(* IEC 61131-3 sources: TIA2AX/tests/V18/test_projects/expected/HW_2000528_ST43/PLC_4.3, 7 files *)

(* ---- HwIdentifiers.st ---- *)
TYPE
	HwIdentifiers : WORD
	(
		PLC_4_3_Rail_0 :=	WORD#256,
		PLC_4_3 :=	WORD#48,
		PLC_4_3_Card_reader_writer_1 :=	WORD#51,
		PLC_4_3_CPU_display_1 :=	WORD#54,
		PLC_4_3_OPC_UA_1 :=	WORD#117,
		PLC_4_3_PROFINET_interface_1 :=	WORD#64,
		PLC_4_3_PROFINET_interface_1_Port_1 :=	WORD#65,
		PLC_4_3_PROFINET_interface_1_Port_2 :=	WORD#66,
		PLC_4_3_PROFINET_interface_2 :=	WORD#72,
		PLC_4_3_PROFINET_interface_2_Port_1 :=	WORD#73,
		wp4_3_dm262_l_Rack :=	WORD#270,
		wp4_3_dm262_l :=	WORD#258,
		wp4_3_dm262_l_Interface :=	WORD#259,
		wp4_3_dm262_l_Interface_Port_1 :=	WORD#260,
		wp4_3_dm262_l_DataMan_260 :=	WORD#261,
		wp4_3_dm262_l_Acquisition_Control_1 :=	WORD#262,
		wp4_3_dm262_l_Acquisition_Status_1 :=	WORD#263,
		wp4_3_dm262_l_Results_Control_1 :=	WORD#264,
		wp4_3_dm262_l_Results_Status_1 :=	WORD#265,
		wp4_3_dm262_l_Soft_Event_Control_1 :=	WORD#266,
		wp4_3_dm262_l_User_Data_64_bytes_1 :=	WORD#267,
		wp4_3_dm262_l_Result_Data_64_bytes_1 :=	WORD#268,
		ET_200SP_ST43_Rack_0 :=	WORD#278,
		ET_200SP_ST43 :=	WORD#279,
		ET_200SP_ST43_ET_200SP_ST43 :=	WORD#280,
		ET_200SP_ST43_PROFINET_interface :=	WORD#281,
		ET_200SP_ST43_PROFINET_interface_Port_1 :=	WORD#283,
		ET_200SP_ST43_PROFINET_interface_Port_2 :=	WORD#282,
		ET_200SP_ST43_BA_2xRJ45 :=	WORD#283,
		ET_200SP_ST43_A3 :=	WORD#284,
		ET_200SP_ST43_A4 :=	WORD#285,
		ET_200SP_ST43_A5 :=	WORD#286,
		ET_200SP_ST43_DI_16x24VDC_ST_1 :=	WORD#287,
		ET_200SP_ST43_DI_16x24VDC_ST_2 :=	WORD#288,
		ET_200SP_ST43_DI_16x24VDC_ST_3 :=	WORD#289,
		ET_200SP_ST43_DI_16x24VDC_ST_4 :=	WORD#290,
		ET_200SP_ST43_DQ_16x24VDC_0_5A_ST_1 :=	WORD#291,
		ET_200SP_ST43_DQ_16x24VDC_0_5A_ST_2 :=	WORD#292,
		ET_200SP_ST43_TM_Pulse_2x24V_1 :=	WORD#271,
		ET_200SP_ST43_TM_Pulse_2x24V_2 :=	WORD#272,
		ET_200SP_ST43_TM_Pulse_2x24V_3 :=	WORD#273,
		ET_200SP_ST43_TM_Pulse_2x24V_4 :=	WORD#274,
		ET_200SP_ST43_TM_Pulse_2x24V_5 :=	WORD#275,
		ET_200SP_ST43_Server_module_1 :=	WORD#276,
		wp4_3_dm262_r_Rack :=	WORD#294,
		wp4_3_dm262_r :=	WORD#295,
		wp4_3_dm262_r_Interface :=	WORD#296,
		wp4_3_dm262_r_Interface_Port_1 :=	WORD#297,
		wp4_3_dm262_r_DataMan_260 :=	WORD#298,
		wp4_3_dm262_r_Acquisition_Control_1 :=	WORD#299,
		wp4_3_dm262_r_Acquisition_Status_1 :=	WORD#300,
		wp4_3_dm262_r_Results_Control_1 :=	WORD#301,
		wp4_3_dm262_r_Results_Status_1 :=	WORD#302,
		wp4_3_dm262_r_Soft_Event_Control_1 :=	WORD#303,
		wp4_3_dm262_r_User_Data_64_bytes_1 :=	WORD#304,
		wp4_3_dm262_r_Result_Data_64_bytes_1 :=	WORD#305,
		CPX_ST43_PN_IO_Interface :=	WORD#309,
		CPX_ST43_PN_IO_Interface_Port_1 :=	WORD#310,
		CPX_ST43_PN_IO_Interface_Port_2 :=	WORD#311,
		CPX_ST43_CPX_Rev_30 :=	WORD#312,
		CPX_ST43_FB33_PNIO_Module_1 :=	WORD#313,
		CPX_ST43_MPA1S_VMPA1_FB_EMS_8_8DO_1 :=	WORD#314,
		CPX_ST43_MPA1G_VMPA1_FB_EMG_8_8DO_1 :=	WORD#315,
		CPX_ST43_MPA1G_VMPA1_FB_EMG_8_8DO_2 :=	WORD#316,
		CPX_ST43_MPA1G_VMPA1_FB_EMG_8_8DO_3 :=	WORD#317,
		CPX_ST43_MPA1G_VMPA1_FB_EMG_8_8DO_4 :=	WORD#318,
		CPX_ST43_MPA1G_VMPA1_FB_EMG_8_8DO_5 :=	WORD#319,
		NONE:= WORD#0
	);
END_TYPE

(* ---- HwInputs.st ---- *)
TYPE
	HwInputs : STRUCT
		wp4_3_dm262_l_Acquisition_Status_1 AT %B317 : ARRAY[0..2] OF BYTE;
		wp4_3_dm262_l_Results_Status_1 AT %B301 : BYTE;
		wp4_3_dm262_l_Soft_Event_Control_1 AT %B302 : BYTE;
		wp4_3_dm262_l_Result_Data_64_bytes_1 AT %B503 : ARRAY[0..71] OF BYTE;
		ET_200SP_ST43_A3 AT %B88 : ARRAY[0..7] OF BYTE;
		ET_200SP_ST43_A4 AT %B96 : ARRAY[0..7] OF BYTE;
		ET_200SP_ST43_A5 AT %B104 : ARRAY[0..7] OF BYTE;
		ET_200SP_ST43_DI_16x24VDC_ST_1 AT %B0 : WORD;
		ET_200SP_ST43_DI_16x24VDC_ST_2 AT %B2 : WORD;
		ET_200SP_ST43_DI_16x24VDC_ST_3 AT %B4 : WORD;
		ET_200SP_ST43_DI_16x24VDC_ST_4 AT %B6 : WORD;
		ET_200SP_ST43_TM_Pulse_2x24V_1 AT %B8 : ARRAY[0..15] OF BYTE;
		ET_200SP_ST43_TM_Pulse_2x24V_2 AT %B24 : ARRAY[0..15] OF BYTE;
		ET_200SP_ST43_TM_Pulse_2x24V_3 AT %B40 : ARRAY[0..15] OF BYTE;
		ET_200SP_ST43_TM_Pulse_2x24V_4 AT %B56 : ARRAY[0..15] OF BYTE;
		ET_200SP_ST43_TM_Pulse_2x24V_5 AT %B72 : ARRAY[0..15] OF BYTE;
		wp4_3_dm262_r_Acquisition_Status_1 AT %B281 : ARRAY[0..2] OF BYTE;
		wp4_3_dm262_r_Results_Status_1 AT %B207 : BYTE;
		wp4_3_dm262_r_Soft_Event_Control_1 AT %B208 : BYTE;
		wp4_3_dm262_r_Result_Data_64_bytes_1 AT %B209 : ARRAY[0..71] OF BYTE;
	END_STRUCT;
END_TYPE

(* ---- HwOutputs.st ---- *)
TYPE
	HwOutputs : STRUCT
		wp4_3_dm262_l_Acquisition_Control_1 AT %B300 : BYTE;
		wp4_3_dm262_l_Results_Control_1 AT %B301 : BYTE;
		wp4_3_dm262_l_Soft_Event_Control_1 AT %B302 : BYTE;
		wp4_3_dm262_l_User_Data_64_bytes_1 AT %B303 : ARRAY[0..67] OF BYTE;
		ET_200SP_ST43_DQ_16x24VDC_0_5A_ST_1 AT %B0 : WORD;
		ET_200SP_ST43_DQ_16x24VDC_0_5A_ST_2 AT %B2 : WORD;
		ET_200SP_ST43_TM_Pulse_2x24V_1 AT %B4 : ARRAY[0..23] OF BYTE;
		ET_200SP_ST43_TM_Pulse_2x24V_2 AT %B56 : ARRAY[0..23] OF BYTE;
		ET_200SP_ST43_TM_Pulse_2x24V_3 AT %B80 : ARRAY[0..23] OF BYTE;
		ET_200SP_ST43_TM_Pulse_2x24V_4 AT %B104 : ARRAY[0..23] OF BYTE;
		ET_200SP_ST43_TM_Pulse_2x24V_5 AT %B128 : ARRAY[0..23] OF BYTE;
		wp4_3_dm262_r_Acquisition_Control_1 AT %B400 : BYTE;
		wp4_3_dm262_r_Results_Control_1 AT %B401 : BYTE;
		wp4_3_dm262_r_Soft_Event_Control_1 AT %B402 : BYTE;
		wp4_3_dm262_r_User_Data_64_bytes_1 AT %B403 : ARRAY[0..67] OF BYTE;
		CPX_ST43_MPA1S_VMPA1_FB_EMS_8_8DO_1 AT %B50 : BYTE;
		CPX_ST43_MPA1G_VMPA1_FB_EMG_8_8DO_1 AT %B51 : BYTE;
		CPX_ST43_MPA1G_VMPA1_FB_EMG_8_8DO_2 AT %B52 : BYTE;
		CPX_ST43_MPA1G_VMPA1_FB_EMG_8_8DO_3 AT %B53 : BYTE;
		CPX_ST43_MPA1G_VMPA1_FB_EMG_8_8DO_4 AT %B54 : BYTE;
		CPX_ST43_MPA1G_VMPA1_FB_EMG_8_8DO_5 AT %B55 : BYTE;
	END_STRUCT;
END_TYPE

(* ---- PlcInputs.st ---- *)
TYPE
	PlcInputs : STRUCT
		wp4_3_dm262_l_Acquisition_Status_1 : ARRAY[0..2] OF BYTE;
		wp4_3_dm262_l_Results_Status_1 : BYTE;
		wp4_3_dm262_l_Soft_Event_Control_1 : BYTE;
		wp4_3_dm262_l_Result_Data_64_bytes_1 : ARRAY[0..71] OF BYTE;
		ET_200SP_ST43_A3 : ARRAY[0..7] OF BYTE;
		ET_200SP_ST43_A4 : ARRAY[0..7] OF BYTE;
		ET_200SP_ST43_A5 : ARRAY[0..7] OF BYTE;
		ET_200SP_ST43_DI_16x24VDC_ST_1 : WORD;
		ET_200SP_ST43_DI_16x24VDC_ST_2 : WORD;
		ET_200SP_ST43_DI_16x24VDC_ST_3 : WORD;
		ET_200SP_ST43_DI_16x24VDC_ST_4 : WORD;
		ET_200SP_ST43_TM_Pulse_2x24V_1 : ARRAY[0..15] OF BYTE;
		ET_200SP_ST43_TM_Pulse_2x24V_2 : ARRAY[0..15] OF BYTE;
		ET_200SP_ST43_TM_Pulse_2x24V_3 : ARRAY[0..15] OF BYTE;
		ET_200SP_ST43_TM_Pulse_2x24V_4 : ARRAY[0..15] OF BYTE;
		ET_200SP_ST43_TM_Pulse_2x24V_5 : ARRAY[0..15] OF BYTE;
		wp4_3_dm262_r_Acquisition_Status_1 : ARRAY[0..2] OF BYTE;
		wp4_3_dm262_r_Results_Status_1 : BYTE;
		wp4_3_dm262_r_Soft_Event_Control_1 : BYTE;
		wp4_3_dm262_r_Result_Data_64_bytes_1 : ARRAY[0..71] OF BYTE;
	END_STRUCT;
END_TYPE

(* ---- PlcOutputs.st ---- *)
TYPE
	PlcOutputs : STRUCT
		wp4_3_dm262_l_Acquisition_Control_1 : BYTE;
		wp4_3_dm262_l_Results_Control_1 : BYTE;
		wp4_3_dm262_l_Soft_Event_Control_1 : BYTE;
		wp4_3_dm262_l_User_Data_64_bytes_1 : ARRAY[0..67] OF BYTE;
		ET_200SP_ST43_DQ_16x24VDC_0_5A_ST_1 : WORD;
		ET_200SP_ST43_DQ_16x24VDC_0_5A_ST_2 : WORD;
		ET_200SP_ST43_TM_Pulse_2x24V_1 : ARRAY[0..23] OF BYTE;
		ET_200SP_ST43_TM_Pulse_2x24V_2 : ARRAY[0..23] OF BYTE;
		ET_200SP_ST43_TM_Pulse_2x24V_3 : ARRAY[0..23] OF BYTE;
		ET_200SP_ST43_TM_Pulse_2x24V_4 : ARRAY[0..23] OF BYTE;
		ET_200SP_ST43_TM_Pulse_2x24V_5 : ARRAY[0..23] OF BYTE;
		wp4_3_dm262_r_Acquisition_Control_1 : BYTE;
		wp4_3_dm262_r_Results_Control_1 : BYTE;
		wp4_3_dm262_r_Soft_Event_Control_1 : BYTE;
		wp4_3_dm262_r_User_Data_64_bytes_1 : ARRAY[0..67] OF BYTE;
		CPX_ST43_MPA1S_VMPA1_FB_EMS_8_8DO_1 : BYTE;
		CPX_ST43_MPA1G_VMPA1_FB_EMG_8_8DO_1 : BYTE;
		CPX_ST43_MPA1G_VMPA1_FB_EMG_8_8DO_2 : BYTE;
		CPX_ST43_MPA1G_VMPA1_FB_EMG_8_8DO_3 : BYTE;
		CPX_ST43_MPA1G_VMPA1_FB_EMG_8_8DO_4 : BYTE;
		CPX_ST43_MPA1G_VMPA1_FB_EMG_8_8DO_5 : BYTE;
	END_STRUCT;
END_TYPE

(* ---- CopyInputs.st ---- *)
FUNCTION CopyInputs
	VAR_EXTERNAL
		HwInputs : HwInputs;
		PlcInputs : PlcInputs;
	END_VAR
	PlcInputs.wp4_3_dm262_l_Acquisition_Status_1[0] := HwInputs.wp4_3_dm262_l_Acquisition_Status_1[0];
	PlcInputs.wp4_3_dm262_l_Acquisition_Status_1[1] := HwInputs.wp4_3_dm262_l_Acquisition_Status_1[1];
	PlcInputs.wp4_3_dm262_l_Acquisition_Status_1[2] := HwInputs.wp4_3_dm262_l_Acquisition_Status_1[2];
	PlcInputs.wp4_3_dm262_l_Results_Status_1 := HwInputs.wp4_3_dm262_l_Results_Status_1;
	PlcInputs.wp4_3_dm262_l_Soft_Event_Control_1 := HwInputs.wp4_3_dm262_l_Soft_Event_Control_1;
	PlcInputs.wp4_3_dm262_l_Result_Data_64_bytes_1[0] := HwInputs.wp4_3_dm262_l_Result_Data_64_bytes_1[0];
	PlcInputs.wp4_3_dm262_l_Result_Data_64_bytes_1[1] := HwInputs.wp4_3_dm262_l_Result_Data_64_bytes_1[1];
	PlcInputs.wp4_3_dm262_l_Result_Data_64_bytes_1[2] := HwInputs.wp4_3_dm262_l_Result_Data_64_bytes_1[2];
	PlcInputs.wp4_3_dm262_l_Result_Data_64_bytes_1[3] := HwInputs.wp4_3_dm262_l_Result_Data_64_bytes_1[3];
	PlcInputs.wp4_3_dm262_l_Result_Data_64_bytes_1[4] := HwInputs.wp4_3_dm262_l_Result_Data_64_bytes_1[4];
	PlcInputs.wp4_3_dm262_l_Result_Data_64_bytes_1[5] := HwInputs.wp4_3_dm262_l_Result_Data_64_bytes_1[5];
	PlcInputs.wp4_3_dm262_l_Result_Data_64_bytes_1[6] := HwInputs.wp4_3_dm262_l_Result_Data_64_bytes_1[6];
	PlcInputs.wp4_3_dm262_l_Result_Data_64_bytes_1[7] := HwInputs.wp4_3_dm262_l_Result_Data_64_bytes_1[7];
	PlcInputs.wp4_3_dm262_l_Result_Data_64_bytes_1[8] := HwInputs.wp4_3_dm262_l_Result_Data_64_bytes_1[8];
	PlcInputs.wp4_3_dm262_l_Result_Data_64_bytes_1[9] := HwInputs.wp4_3_dm262_l_Result_Data_64_bytes_1[9];
	PlcInputs.wp4_3_dm262_l_Result_Data_64_bytes_1[10] := HwInputs.wp4_3_dm262_l_Result_Data_64_bytes_1[10];
	PlcInputs.wp4_3_dm262_l_Result_Data_64_bytes_1[11] := HwInputs.wp4_3_dm262_l_Result_Data_64_bytes_1[11];
	PlcInputs.wp4_3_dm262_l_Result_Data_64_bytes_1[12] := HwInputs.wp4_3_dm262_l_Result_Data_64_bytes_1[12];
	PlcInputs.wp4_3_dm262_l_Result_Data_64_bytes_1[13] := HwInputs.wp4_3_dm262_l_Result_Data_64_bytes_1[13];
	PlcInputs.wp4_3_dm262_l_Result_Data_64_bytes_1[14] := HwInputs.wp4_3_dm262_l_Result_Data_64_bytes_1[14];
	PlcInputs.wp4_3_dm262_l_Result_Data_64_bytes_1[15] := HwInputs.wp4_3_dm262_l_Result_Data_64_bytes_1[15];
	PlcInputs.wp4_3_dm262_l_Result_Data_64_bytes_1[16] := HwInputs.wp4_3_dm262_l_Result_Data_64_bytes_1[16];
	PlcInputs.wp4_3_dm262_l_Result_Data_64_bytes_1[17] := HwInputs.wp4_3_dm262_l_Result_Data_64_bytes_1[17];
	PlcInputs.wp4_3_dm262_l_Result_Data_64_bytes_1[18] := HwInputs.wp4_3_dm262_l_Result_Data_64_bytes_1[18];
	PlcInputs.wp4_3_dm262_l_Result_Data_64_bytes_1[19] := HwInputs.wp4_3_dm262_l_Result_Data_64_bytes_1[19];
	PlcInputs.wp4_3_dm262_l_Result_Data_64_bytes_1[20] := HwInputs.wp4_3_dm262_l_Result_Data_64_bytes_1[20];
	PlcInputs.wp4_3_dm262_l_Result_Data_64_bytes_1[21] := HwInputs.wp4_3_dm262_l_Result_Data_64_bytes_1[21];
	PlcInputs.wp4_3_dm262_l_Result_Data_64_bytes_1[22] := HwInputs.wp4_3_dm262_l_Result_Data_64_bytes_1[22];
	PlcInputs.wp4_3_dm262_l_Result_Data_64_bytes_1[23] := HwInputs.wp4_3_dm262_l_Result_Data_64_bytes_1[23];
	PlcInputs.wp4_3_dm262_l_Result_Data_64_bytes_1[24] := HwInputs.wp4_3_dm262_l_Result_Data_64_bytes_1[24];
	PlcInputs.wp4_3_dm262_l_Result_Data_64_bytes_1[25] := HwInputs.wp4_3_dm262_l_Result_Data_64_bytes_1[25];
	PlcInputs.wp4_3_dm262_l_Result_Data_64_bytes_1[26] := HwInputs.wp4_3_dm262_l_Result_Data_64_bytes_1[26];
	PlcInputs.wp4_3_dm262_l_Result_Data_64_bytes_1[27] := HwInputs.wp4_3_dm262_l_Result_Data_64_bytes_1[27];
	PlcInputs.wp4_3_dm262_l_Result_Data_64_bytes_1[28] := HwInputs.wp4_3_dm262_l_Result_Data_64_bytes_1[28];
	PlcInputs.wp4_3_dm262_l_Result_Data_64_bytes_1[29] := HwInputs.wp4_3_dm262_l_Result_Data_64_bytes_1[29];
	PlcInputs.wp4_3_dm262_l_Result_Data_64_bytes_1[30] := HwInputs.wp4_3_dm262_l_Result_Data_64_bytes_1[30];
	PlcInputs.wp4_3_dm262_l_Result_Data_64_bytes_1[31] := HwInputs.wp4_3_dm262_l_Result_Data_64_bytes_1[31];
	PlcInputs.wp4_3_dm262_l_Result_Data_64_bytes_1[32] := HwInputs.wp4_3_dm262_l_Result_Data_64_bytes_1[32];
	PlcInputs.wp4_3_dm262_l_Result_Data_64_bytes_1[33] := HwInputs.wp4_3_dm262_l_Result_Data_64_bytes_1[33];
	PlcInputs.wp4_3_dm262_l_Result_Data_64_bytes_1[34] := HwInputs.wp4_3_dm262_l_Result_Data_64_bytes_1[34];
	PlcInputs.wp4_3_dm262_l_Result_Data_64_bytes_1[35] := HwInputs.wp4_3_dm262_l_Result_Data_64_bytes_1[35];
	PlcInputs.wp4_3_dm262_l_Result_Data_64_bytes_1[36] := HwInputs.wp4_3_dm262_l_Result_Data_64_bytes_1[36];
	PlcInputs.wp4_3_dm262_l_Result_Data_64_bytes_1[37] := HwInputs.wp4_3_dm262_l_Result_Data_64_bytes_1[37];
	PlcInputs.wp4_3_dm262_l_Result_Data_64_bytes_1[38] := HwInputs.wp4_3_dm262_l_Result_Data_64_bytes_1[38];
	PlcInputs.wp4_3_dm262_l_Result_Data_64_bytes_1[39] := HwInputs.wp4_3_dm262_l_Result_Data_64_bytes_1[39];
	PlcInputs.wp4_3_dm262_l_Result_Data_64_bytes_1[40] := HwInputs.wp4_3_dm262_l_Result_Data_64_bytes_1[40];
	PlcInputs.wp4_3_dm262_l_Result_Data_64_bytes_1[41] := HwInputs.wp4_3_dm262_l_Result_Data_64_bytes_1[41];
	PlcInputs.wp4_3_dm262_l_Result_Data_64_bytes_1[42] := HwInputs.wp4_3_dm262_l_Result_Data_64_bytes_1[42];
	PlcInputs.wp4_3_dm262_l_Result_Data_64_bytes_1[43] := HwInputs.wp4_3_dm262_l_Result_Data_64_bytes_1[43];
	PlcInputs.wp4_3_dm262_l_Result_Data_64_bytes_1[44] := HwInputs.wp4_3_dm262_l_Result_Data_64_bytes_1[44];
	PlcInputs.wp4_3_dm262_l_Result_Data_64_bytes_1[45] := HwInputs.wp4_3_dm262_l_Result_Data_64_bytes_1[45];
	PlcInputs.wp4_3_dm262_l_Result_Data_64_bytes_1[46] := HwInputs.wp4_3_dm262_l_Result_Data_64_bytes_1[46];
	PlcInputs.wp4_3_dm262_l_Result_Data_64_bytes_1[47] := HwInputs.wp4_3_dm262_l_Result_Data_64_bytes_1[47];
	PlcInputs.wp4_3_dm262_l_Result_Data_64_bytes_1[48] := HwInputs.wp4_3_dm262_l_Result_Data_64_bytes_1[48];
	PlcInputs.wp4_3_dm262_l_Result_Data_64_bytes_1[49] := HwInputs.wp4_3_dm262_l_Result_Data_64_bytes_1[49];
	PlcInputs.wp4_3_dm262_l_Result_Data_64_bytes_1[50] := HwInputs.wp4_3_dm262_l_Result_Data_64_bytes_1[50];
	PlcInputs.wp4_3_dm262_l_Result_Data_64_bytes_1[51] := HwInputs.wp4_3_dm262_l_Result_Data_64_bytes_1[51];
	PlcInputs.wp4_3_dm262_l_Result_Data_64_bytes_1[52] := HwInputs.wp4_3_dm262_l_Result_Data_64_bytes_1[52];
	PlcInputs.wp4_3_dm262_l_Result_Data_64_bytes_1[53] := HwInputs.wp4_3_dm262_l_Result_Data_64_bytes_1[53];
	PlcInputs.wp4_3_dm262_l_Result_Data_64_bytes_1[54] := HwInputs.wp4_3_dm262_l_Result_Data_64_bytes_1[54];
	PlcInputs.wp4_3_dm262_l_Result_Data_64_bytes_1[55] := HwInputs.wp4_3_dm262_l_Result_Data_64_bytes_1[55];
	PlcInputs.wp4_3_dm262_l_Result_Data_64_bytes_1[56] := HwInputs.wp4_3_dm262_l_Result_Data_64_bytes_1[56];
	PlcInputs.wp4_3_dm262_l_Result_Data_64_bytes_1[57] := HwInputs.wp4_3_dm262_l_Result_Data_64_bytes_1[57];
	PlcInputs.wp4_3_dm262_l_Result_Data_64_bytes_1[58] := HwInputs.wp4_3_dm262_l_Result_Data_64_bytes_1[58];
	PlcInputs.wp4_3_dm262_l_Result_Data_64_bytes_1[59] := HwInputs.wp4_3_dm262_l_Result_Data_64_bytes_1[59];
	PlcInputs.wp4_3_dm262_l_Result_Data_64_bytes_1[60] := HwInputs.wp4_3_dm262_l_Result_Data_64_bytes_1[60];
	PlcInputs.wp4_3_dm262_l_Result_Data_64_bytes_1[61] := HwInputs.wp4_3_dm262_l_Result_Data_64_bytes_1[61];
	PlcInputs.wp4_3_dm262_l_Result_Data_64_bytes_1[62] := HwInputs.wp4_3_dm262_l_Result_Data_64_bytes_1[62];
	PlcInputs.wp4_3_dm262_l_Result_Data_64_bytes_1[63] := HwInputs.wp4_3_dm262_l_Result_Data_64_bytes_1[63];
	PlcInputs.wp4_3_dm262_l_Result_Data_64_bytes_1[64] := HwInputs.wp4_3_dm262_l_Result_Data_64_bytes_1[64];
	PlcInputs.wp4_3_dm262_l_Result_Data_64_bytes_1[65] := HwInputs.wp4_3_dm262_l_Result_Data_64_bytes_1[65];
	PlcInputs.wp4_3_dm262_l_Result_Data_64_bytes_1[66] := HwInputs.wp4_3_dm262_l_Result_Data_64_bytes_1[66];
	PlcInputs.wp4_3_dm262_l_Result_Data_64_bytes_1[67] := HwInputs.wp4_3_dm262_l_Result_Data_64_bytes_1[67];
	PlcInputs.wp4_3_dm262_l_Result_Data_64_bytes_1[68] := HwInputs.wp4_3_dm262_l_Result_Data_64_bytes_1[68];
	PlcInputs.wp4_3_dm262_l_Result_Data_64_bytes_1[69] := HwInputs.wp4_3_dm262_l_Result_Data_64_bytes_1[69];
	PlcInputs.wp4_3_dm262_l_Result_Data_64_bytes_1[70] := HwInputs.wp4_3_dm262_l_Result_Data_64_bytes_1[70];
	PlcInputs.wp4_3_dm262_l_Result_Data_64_bytes_1[71] := HwInputs.wp4_3_dm262_l_Result_Data_64_bytes_1[71];
	PlcInputs.ET_200SP_ST43_A3[0] := HwInputs.ET_200SP_ST43_A3[0];
	PlcInputs.ET_200SP_ST43_A3[1] := HwInputs.ET_200SP_ST43_A3[1];
	PlcInputs.ET_200SP_ST43_A3[2] := HwInputs.ET_200SP_ST43_A3[2];
	PlcInputs.ET_200SP_ST43_A3[3] := HwInputs.ET_200SP_ST43_A3[3];
	PlcInputs.ET_200SP_ST43_A3[4] := HwInputs.ET_200SP_ST43_A3[4];
	PlcInputs.ET_200SP_ST43_A3[5] := HwInputs.ET_200SP_ST43_A3[5];
	PlcInputs.ET_200SP_ST43_A3[6] := HwInputs.ET_200SP_ST43_A3[6];
	PlcInputs.ET_200SP_ST43_A3[7] := HwInputs.ET_200SP_ST43_A3[7];
	PlcInputs.ET_200SP_ST43_A4[0] := HwInputs.ET_200SP_ST43_A4[0];
	PlcInputs.ET_200SP_ST43_A4[1] := HwInputs.ET_200SP_ST43_A4[1];
	PlcInputs.ET_200SP_ST43_A4[2] := HwInputs.ET_200SP_ST43_A4[2];
	PlcInputs.ET_200SP_ST43_A4[3] := HwInputs.ET_200SP_ST43_A4[3];
	PlcInputs.ET_200SP_ST43_A4[4] := HwInputs.ET_200SP_ST43_A4[4];
	PlcInputs.ET_200SP_ST43_A4[5] := HwInputs.ET_200SP_ST43_A4[5];
	PlcInputs.ET_200SP_ST43_A4[6] := HwInputs.ET_200SP_ST43_A4[6];
	PlcInputs.ET_200SP_ST43_A4[7] := HwInputs.ET_200SP_ST43_A4[7];
	PlcInputs.ET_200SP_ST43_A5[0] := HwInputs.ET_200SP_ST43_A5[0];
	PlcInputs.ET_200SP_ST43_A5[1] := HwInputs.ET_200SP_ST43_A5[1];
	PlcInputs.ET_200SP_ST43_A5[2] := HwInputs.ET_200SP_ST43_A5[2];
	PlcInputs.ET_200SP_ST43_A5[3] := HwInputs.ET_200SP_ST43_A5[3];
	PlcInputs.ET_200SP_ST43_A5[4] := HwInputs.ET_200SP_ST43_A5[4];
	PlcInputs.ET_200SP_ST43_A5[5] := HwInputs.ET_200SP_ST43_A5[5];
	PlcInputs.ET_200SP_ST43_A5[6] := HwInputs.ET_200SP_ST43_A5[6];
	PlcInputs.ET_200SP_ST43_A5[7] := HwInputs.ET_200SP_ST43_A5[7];
	PlcInputs.ET_200SP_ST43_DI_16x24VDC_ST_1 := HwInputs.ET_200SP_ST43_DI_16x24VDC_ST_1;
	PlcInputs.ET_200SP_ST43_DI_16x24VDC_ST_2 := HwInputs.ET_200SP_ST43_DI_16x24VDC_ST_2;
	PlcInputs.ET_200SP_ST43_DI_16x24VDC_ST_3 := HwInputs.ET_200SP_ST43_DI_16x24VDC_ST_3;
	PlcInputs.ET_200SP_ST43_DI_16x24VDC_ST_4 := HwInputs.ET_200SP_ST43_DI_16x24VDC_ST_4;
	PlcInputs.ET_200SP_ST43_TM_Pulse_2x24V_1[0] := HwInputs.ET_200SP_ST43_TM_Pulse_2x24V_1[0];
	PlcInputs.ET_200SP_ST43_TM_Pulse_2x24V_1[1] := HwInputs.ET_200SP_ST43_TM_Pulse_2x24V_1[1];
	PlcInputs.ET_200SP_ST43_TM_Pulse_2x24V_1[2] := HwInputs.ET_200SP_ST43_TM_Pulse_2x24V_1[2];
	PlcInputs.ET_200SP_ST43_TM_Pulse_2x24V_1[3] := HwInputs.ET_200SP_ST43_TM_Pulse_2x24V_1[3];
	PlcInputs.ET_200SP_ST43_TM_Pulse_2x24V_1[4] := HwInputs.ET_200SP_ST43_TM_Pulse_2x24V_1[4];
	PlcInputs.ET_200SP_ST43_TM_Pulse_2x24V_1[5] := HwInputs.ET_200SP_ST43_TM_Pulse_2x24V_1[5];
	PlcInputs.ET_200SP_ST43_TM_Pulse_2x24V_1[6] := HwInputs.ET_200SP_ST43_TM_Pulse_2x24V_1[6];
	PlcInputs.ET_200SP_ST43_TM_Pulse_2x24V_1[7] := HwInputs.ET_200SP_ST43_TM_Pulse_2x24V_1[7];
	PlcInputs.ET_200SP_ST43_TM_Pulse_2x24V_1[8] := HwInputs.ET_200SP_ST43_TM_Pulse_2x24V_1[8];
	PlcInputs.ET_200SP_ST43_TM_Pulse_2x24V_1[9] := HwInputs.ET_200SP_ST43_TM_Pulse_2x24V_1[9];
	PlcInputs.ET_200SP_ST43_TM_Pulse_2x24V_1[10] := HwInputs.ET_200SP_ST43_TM_Pulse_2x24V_1[10];
	PlcInputs.ET_200SP_ST43_TM_Pulse_2x24V_1[11] := HwInputs.ET_200SP_ST43_TM_Pulse_2x24V_1[11];
	PlcInputs.ET_200SP_ST43_TM_Pulse_2x24V_1[12] := HwInputs.ET_200SP_ST43_TM_Pulse_2x24V_1[12];
	PlcInputs.ET_200SP_ST43_TM_Pulse_2x24V_1[13] := HwInputs.ET_200SP_ST43_TM_Pulse_2x24V_1[13];
	PlcInputs.ET_200SP_ST43_TM_Pulse_2x24V_1[14] := HwInputs.ET_200SP_ST43_TM_Pulse_2x24V_1[14];
	PlcInputs.ET_200SP_ST43_TM_Pulse_2x24V_1[15] := HwInputs.ET_200SP_ST43_TM_Pulse_2x24V_1[15];
	PlcInputs.ET_200SP_ST43_TM_Pulse_2x24V_2[0] := HwInputs.ET_200SP_ST43_TM_Pulse_2x24V_2[0];
	PlcInputs.ET_200SP_ST43_TM_Pulse_2x24V_2[1] := HwInputs.ET_200SP_ST43_TM_Pulse_2x24V_2[1];
	PlcInputs.ET_200SP_ST43_TM_Pulse_2x24V_2[2] := HwInputs.ET_200SP_ST43_TM_Pulse_2x24V_2[2];
	PlcInputs.ET_200SP_ST43_TM_Pulse_2x24V_2[3] := HwInputs.ET_200SP_ST43_TM_Pulse_2x24V_2[3];
	PlcInputs.ET_200SP_ST43_TM_Pulse_2x24V_2[4] := HwInputs.ET_200SP_ST43_TM_Pulse_2x24V_2[4];
	PlcInputs.ET_200SP_ST43_TM_Pulse_2x24V_2[5] := HwInputs.ET_200SP_ST43_TM_Pulse_2x24V_2[5];
	PlcInputs.ET_200SP_ST43_TM_Pulse_2x24V_2[6] := HwInputs.ET_200SP_ST43_TM_Pulse_2x24V_2[6];
	PlcInputs.ET_200SP_ST43_TM_Pulse_2x24V_2[7] := HwInputs.ET_200SP_ST43_TM_Pulse_2x24V_2[7];
	PlcInputs.ET_200SP_ST43_TM_Pulse_2x24V_2[8] := HwInputs.ET_200SP_ST43_TM_Pulse_2x24V_2[8];
	PlcInputs.ET_200SP_ST43_TM_Pulse_2x24V_2[9] := HwInputs.ET_200SP_ST43_TM_Pulse_2x24V_2[9];
	PlcInputs.ET_200SP_ST43_TM_Pulse_2x24V_2[10] := HwInputs.ET_200SP_ST43_TM_Pulse_2x24V_2[10];
	PlcInputs.ET_200SP_ST43_TM_Pulse_2x24V_2[11] := HwInputs.ET_200SP_ST43_TM_Pulse_2x24V_2[11];
	PlcInputs.ET_200SP_ST43_TM_Pulse_2x24V_2[12] := HwInputs.ET_200SP_ST43_TM_Pulse_2x24V_2[12];
	PlcInputs.ET_200SP_ST43_TM_Pulse_2x24V_2[13] := HwInputs.ET_200SP_ST43_TM_Pulse_2x24V_2[13];
	PlcInputs.ET_200SP_ST43_TM_Pulse_2x24V_2[14] := HwInputs.ET_200SP_ST43_TM_Pulse_2x24V_2[14];
	PlcInputs.ET_200SP_ST43_TM_Pulse_2x24V_2[15] := HwInputs.ET_200SP_ST43_TM_Pulse_2x24V_2[15];
	PlcInputs.ET_200SP_ST43_TM_Pulse_2x24V_3[0] := HwInputs.ET_200SP_ST43_TM_Pulse_2x24V_3[0];
	PlcInputs.ET_200SP_ST43_TM_Pulse_2x24V_3[1] := HwInputs.ET_200SP_ST43_TM_Pulse_2x24V_3[1];
	PlcInputs.ET_200SP_ST43_TM_Pulse_2x24V_3[2] := HwInputs.ET_200SP_ST43_TM_Pulse_2x24V_3[2];
	PlcInputs.ET_200SP_ST43_TM_Pulse_2x24V_3[3] := HwInputs.ET_200SP_ST43_TM_Pulse_2x24V_3[3];
	PlcInputs.ET_200SP_ST43_TM_Pulse_2x24V_3[4] := HwInputs.ET_200SP_ST43_TM_Pulse_2x24V_3[4];
	PlcInputs.ET_200SP_ST43_TM_Pulse_2x24V_3[5] := HwInputs.ET_200SP_ST43_TM_Pulse_2x24V_3[5];
	PlcInputs.ET_200SP_ST43_TM_Pulse_2x24V_3[6] := HwInputs.ET_200SP_ST43_TM_Pulse_2x24V_3[6];
	PlcInputs.ET_200SP_ST43_TM_Pulse_2x24V_3[7] := HwInputs.ET_200SP_ST43_TM_Pulse_2x24V_3[7];
	PlcInputs.ET_200SP_ST43_TM_Pulse_2x24V_3[8] := HwInputs.ET_200SP_ST43_TM_Pulse_2x24V_3[8];
	PlcInputs.ET_200SP_ST43_TM_Pulse_2x24V_3[9] := HwInputs.ET_200SP_ST43_TM_Pulse_2x24V_3[9];
	PlcInputs.ET_200SP_ST43_TM_Pulse_2x24V_3[10] := HwInputs.ET_200SP_ST43_TM_Pulse_2x24V_3[10];
	PlcInputs.ET_200SP_ST43_TM_Pulse_2x24V_3[11] := HwInputs.ET_200SP_ST43_TM_Pulse_2x24V_3[11];
	PlcInputs.ET_200SP_ST43_TM_Pulse_2x24V_3[12] := HwInputs.ET_200SP_ST43_TM_Pulse_2x24V_3[12];
	PlcInputs.ET_200SP_ST43_TM_Pulse_2x24V_3[13] := HwInputs.ET_200SP_ST43_TM_Pulse_2x24V_3[13];
	PlcInputs.ET_200SP_ST43_TM_Pulse_2x24V_3[14] := HwInputs.ET_200SP_ST43_TM_Pulse_2x24V_3[14];
	PlcInputs.ET_200SP_ST43_TM_Pulse_2x24V_3[15] := HwInputs.ET_200SP_ST43_TM_Pulse_2x24V_3[15];
	PlcInputs.ET_200SP_ST43_TM_Pulse_2x24V_4[0] := HwInputs.ET_200SP_ST43_TM_Pulse_2x24V_4[0];
	PlcInputs.ET_200SP_ST43_TM_Pulse_2x24V_4[1] := HwInputs.ET_200SP_ST43_TM_Pulse_2x24V_4[1];
	PlcInputs.ET_200SP_ST43_TM_Pulse_2x24V_4[2] := HwInputs.ET_200SP_ST43_TM_Pulse_2x24V_4[2];
	PlcInputs.ET_200SP_ST43_TM_Pulse_2x24V_4[3] := HwInputs.ET_200SP_ST43_TM_Pulse_2x24V_4[3];
	PlcInputs.ET_200SP_ST43_TM_Pulse_2x24V_4[4] := HwInputs.ET_200SP_ST43_TM_Pulse_2x24V_4[4];
	PlcInputs.ET_200SP_ST43_TM_Pulse_2x24V_4[5] := HwInputs.ET_200SP_ST43_TM_Pulse_2x24V_4[5];
	PlcInputs.ET_200SP_ST43_TM_Pulse_2x24V_4[6] := HwInputs.ET_200SP_ST43_TM_Pulse_2x24V_4[6];
	PlcInputs.ET_200SP_ST43_TM_Pulse_2x24V_4[7] := HwInputs.ET_200SP_ST43_TM_Pulse_2x24V_4[7];
	PlcInputs.ET_200SP_ST43_TM_Pulse_2x24V_4[8] := HwInputs.ET_200SP_ST43_TM_Pulse_2x24V_4[8];
	PlcInputs.ET_200SP_ST43_TM_Pulse_2x24V_4[9] := HwInputs.ET_200SP_ST43_TM_Pulse_2x24V_4[9];
	PlcInputs.ET_200SP_ST43_TM_Pulse_2x24V_4[10] := HwInputs.ET_200SP_ST43_TM_Pulse_2x24V_4[10];
	PlcInputs.ET_200SP_ST43_TM_Pulse_2x24V_4[11] := HwInputs.ET_200SP_ST43_TM_Pulse_2x24V_4[11];
	PlcInputs.ET_200SP_ST43_TM_Pulse_2x24V_4[12] := HwInputs.ET_200SP_ST43_TM_Pulse_2x24V_4[12];
	PlcInputs.ET_200SP_ST43_TM_Pulse_2x24V_4[13] := HwInputs.ET_200SP_ST43_TM_Pulse_2x24V_4[13];
	PlcInputs.ET_200SP_ST43_TM_Pulse_2x24V_4[14] := HwInputs.ET_200SP_ST43_TM_Pulse_2x24V_4[14];
	PlcInputs.ET_200SP_ST43_TM_Pulse_2x24V_4[15] := HwInputs.ET_200SP_ST43_TM_Pulse_2x24V_4[15];
	PlcInputs.ET_200SP_ST43_TM_Pulse_2x24V_5[0] := HwInputs.ET_200SP_ST43_TM_Pulse_2x24V_5[0];
	PlcInputs.ET_200SP_ST43_TM_Pulse_2x24V_5[1] := HwInputs.ET_200SP_ST43_TM_Pulse_2x24V_5[1];
	PlcInputs.ET_200SP_ST43_TM_Pulse_2x24V_5[2] := HwInputs.ET_200SP_ST43_TM_Pulse_2x24V_5[2];
	PlcInputs.ET_200SP_ST43_TM_Pulse_2x24V_5[3] := HwInputs.ET_200SP_ST43_TM_Pulse_2x24V_5[3];
	PlcInputs.ET_200SP_ST43_TM_Pulse_2x24V_5[4] := HwInputs.ET_200SP_ST43_TM_Pulse_2x24V_5[4];
	PlcInputs.ET_200SP_ST43_TM_Pulse_2x24V_5[5] := HwInputs.ET_200SP_ST43_TM_Pulse_2x24V_5[5];
	PlcInputs.ET_200SP_ST43_TM_Pulse_2x24V_5[6] := HwInputs.ET_200SP_ST43_TM_Pulse_2x24V_5[6];
	PlcInputs.ET_200SP_ST43_TM_Pulse_2x24V_5[7] := HwInputs.ET_200SP_ST43_TM_Pulse_2x24V_5[7];
	PlcInputs.ET_200SP_ST43_TM_Pulse_2x24V_5[8] := HwInputs.ET_200SP_ST43_TM_Pulse_2x24V_5[8];
	PlcInputs.ET_200SP_ST43_TM_Pulse_2x24V_5[9] := HwInputs.ET_200SP_ST43_TM_Pulse_2x24V_5[9];
	PlcInputs.ET_200SP_ST43_TM_Pulse_2x24V_5[10] := HwInputs.ET_200SP_ST43_TM_Pulse_2x24V_5[10];
	PlcInputs.ET_200SP_ST43_TM_Pulse_2x24V_5[11] := HwInputs.ET_200SP_ST43_TM_Pulse_2x24V_5[11];
	PlcInputs.ET_200SP_ST43_TM_Pulse_2x24V_5[12] := HwInputs.ET_200SP_ST43_TM_Pulse_2x24V_5[12];
	PlcInputs.ET_200SP_ST43_TM_Pulse_2x24V_5[13] := HwInputs.ET_200SP_ST43_TM_Pulse_2x24V_5[13];
	PlcInputs.ET_200SP_ST43_TM_Pulse_2x24V_5[14] := HwInputs.ET_200SP_ST43_TM_Pulse_2x24V_5[14];
	PlcInputs.ET_200SP_ST43_TM_Pulse_2x24V_5[15] := HwInputs.ET_200SP_ST43_TM_Pulse_2x24V_5[15];
	PlcInputs.wp4_3_dm262_r_Acquisition_Status_1[0] := HwInputs.wp4_3_dm262_r_Acquisition_Status_1[0];
	PlcInputs.wp4_3_dm262_r_Acquisition_Status_1[1] := HwInputs.wp4_3_dm262_r_Acquisition_Status_1[1];
	PlcInputs.wp4_3_dm262_r_Acquisition_Status_1[2] := HwInputs.wp4_3_dm262_r_Acquisition_Status_1[2];
	PlcInputs.wp4_3_dm262_r_Results_Status_1 := HwInputs.wp4_3_dm262_r_Results_Status_1;
	PlcInputs.wp4_3_dm262_r_Soft_Event_Control_1 := HwInputs.wp4_3_dm262_r_Soft_Event_Control_1;
	PlcInputs.wp4_3_dm262_r_Result_Data_64_bytes_1[0] := HwInputs.wp4_3_dm262_r_Result_Data_64_bytes_1[0];
	PlcInputs.wp4_3_dm262_r_Result_Data_64_bytes_1[1] := HwInputs.wp4_3_dm262_r_Result_Data_64_bytes_1[1];
	PlcInputs.wp4_3_dm262_r_Result_Data_64_bytes_1[2] := HwInputs.wp4_3_dm262_r_Result_Data_64_bytes_1[2];
	PlcInputs.wp4_3_dm262_r_Result_Data_64_bytes_1[3] := HwInputs.wp4_3_dm262_r_Result_Data_64_bytes_1[3];
	PlcInputs.wp4_3_dm262_r_Result_Data_64_bytes_1[4] := HwInputs.wp4_3_dm262_r_Result_Data_64_bytes_1[4];
	PlcInputs.wp4_3_dm262_r_Result_Data_64_bytes_1[5] := HwInputs.wp4_3_dm262_r_Result_Data_64_bytes_1[5];
	PlcInputs.wp4_3_dm262_r_Result_Data_64_bytes_1[6] := HwInputs.wp4_3_dm262_r_Result_Data_64_bytes_1[6];
	PlcInputs.wp4_3_dm262_r_Result_Data_64_bytes_1[7] := HwInputs.wp4_3_dm262_r_Result_Data_64_bytes_1[7];
	PlcInputs.wp4_3_dm262_r_Result_Data_64_bytes_1[8] := HwInputs.wp4_3_dm262_r_Result_Data_64_bytes_1[8];
	PlcInputs.wp4_3_dm262_r_Result_Data_64_bytes_1[9] := HwInputs.wp4_3_dm262_r_Result_Data_64_bytes_1[9];
	PlcInputs.wp4_3_dm262_r_Result_Data_64_bytes_1[10] := HwInputs.wp4_3_dm262_r_Result_Data_64_bytes_1[10];
	PlcInputs.wp4_3_dm262_r_Result_Data_64_bytes_1[11] := HwInputs.wp4_3_dm262_r_Result_Data_64_bytes_1[11];
	PlcInputs.wp4_3_dm262_r_Result_Data_64_bytes_1[12] := HwInputs.wp4_3_dm262_r_Result_Data_64_bytes_1[12];
	PlcInputs.wp4_3_dm262_r_Result_Data_64_bytes_1[13] := HwInputs.wp4_3_dm262_r_Result_Data_64_bytes_1[13];
	PlcInputs.wp4_3_dm262_r_Result_Data_64_bytes_1[14] := HwInputs.wp4_3_dm262_r_Result_Data_64_bytes_1[14];
	PlcInputs.wp4_3_dm262_r_Result_Data_64_bytes_1[15] := HwInputs.wp4_3_dm262_r_Result_Data_64_bytes_1[15];
	PlcInputs.wp4_3_dm262_r_Result_Data_64_bytes_1[16] := HwInputs.wp4_3_dm262_r_Result_Data_64_bytes_1[16];
	PlcInputs.wp4_3_dm262_r_Result_Data_64_bytes_1[17] := HwInputs.wp4_3_dm262_r_Result_Data_64_bytes_1[17];
	PlcInputs.wp4_3_dm262_r_Result_Data_64_bytes_1[18] := HwInputs.wp4_3_dm262_r_Result_Data_64_bytes_1[18];
	PlcInputs.wp4_3_dm262_r_Result_Data_64_bytes_1[19] := HwInputs.wp4_3_dm262_r_Result_Data_64_bytes_1[19];
	PlcInputs.wp4_3_dm262_r_Result_Data_64_bytes_1[20] := HwInputs.wp4_3_dm262_r_Result_Data_64_bytes_1[20];
	PlcInputs.wp4_3_dm262_r_Result_Data_64_bytes_1[21] := HwInputs.wp4_3_dm262_r_Result_Data_64_bytes_1[21];
	PlcInputs.wp4_3_dm262_r_Result_Data_64_bytes_1[22] := HwInputs.wp4_3_dm262_r_Result_Data_64_bytes_1[22];
	PlcInputs.wp4_3_dm262_r_Result_Data_64_bytes_1[23] := HwInputs.wp4_3_dm262_r_Result_Data_64_bytes_1[23];
	PlcInputs.wp4_3_dm262_r_Result_Data_64_bytes_1[24] := HwInputs.wp4_3_dm262_r_Result_Data_64_bytes_1[24];
	PlcInputs.wp4_3_dm262_r_Result_Data_64_bytes_1[25] := HwInputs.wp4_3_dm262_r_Result_Data_64_bytes_1[25];
	PlcInputs.wp4_3_dm262_r_Result_Data_64_bytes_1[26] := HwInputs.wp4_3_dm262_r_Result_Data_64_bytes_1[26];
	PlcInputs.wp4_3_dm262_r_Result_Data_64_bytes_1[27] := HwInputs.wp4_3_dm262_r_Result_Data_64_bytes_1[27];
	PlcInputs.wp4_3_dm262_r_Result_Data_64_bytes_1[28] := HwInputs.wp4_3_dm262_r_Result_Data_64_bytes_1[28];
	PlcInputs.wp4_3_dm262_r_Result_Data_64_bytes_1[29] := HwInputs.wp4_3_dm262_r_Result_Data_64_bytes_1[29];
	PlcInputs.wp4_3_dm262_r_Result_Data_64_bytes_1[30] := HwInputs.wp4_3_dm262_r_Result_Data_64_bytes_1[30];
	PlcInputs.wp4_3_dm262_r_Result_Data_64_bytes_1[31] := HwInputs.wp4_3_dm262_r_Result_Data_64_bytes_1[31];
	PlcInputs.wp4_3_dm262_r_Result_Data_64_bytes_1[32] := HwInputs.wp4_3_dm262_r_Result_Data_64_bytes_1[32];
	PlcInputs.wp4_3_dm262_r_Result_Data_64_bytes_1[33] := HwInputs.wp4_3_dm262_r_Result_Data_64_bytes_1[33];
	PlcInputs.wp4_3_dm262_r_Result_Data_64_bytes_1[34] := HwInputs.wp4_3_dm262_r_Result_Data_64_bytes_1[34];
	PlcInputs.wp4_3_dm262_r_Result_Data_64_bytes_1[35] := HwInputs.wp4_3_dm262_r_Result_Data_64_bytes_1[35];
	PlcInputs.wp4_3_dm262_r_Result_Data_64_bytes_1[36] := HwInputs.wp4_3_dm262_r_Result_Data_64_bytes_1[36];
	PlcInputs.wp4_3_dm262_r_Result_Data_64_bytes_1[37] := HwInputs.wp4_3_dm262_r_Result_Data_64_bytes_1[37];
	PlcInputs.wp4_3_dm262_r_Result_Data_64_bytes_1[38] := HwInputs.wp4_3_dm262_r_Result_Data_64_bytes_1[38];
	PlcInputs.wp4_3_dm262_r_Result_Data_64_bytes_1[39] := HwInputs.wp4_3_dm262_r_Result_Data_64_bytes_1[39];
	PlcInputs.wp4_3_dm262_r_Result_Data_64_bytes_1[40] := HwInputs.wp4_3_dm262_r_Result_Data_64_bytes_1[40];
	PlcInputs.wp4_3_dm262_r_Result_Data_64_bytes_1[41] := HwInputs.wp4_3_dm262_r_Result_Data_64_bytes_1[41];
	PlcInputs.wp4_3_dm262_r_Result_Data_64_bytes_1[42] := HwInputs.wp4_3_dm262_r_Result_Data_64_bytes_1[42];
	PlcInputs.wp4_3_dm262_r_Result_Data_64_bytes_1[43] := HwInputs.wp4_3_dm262_r_Result_Data_64_bytes_1[43];
	PlcInputs.wp4_3_dm262_r_Result_Data_64_bytes_1[44] := HwInputs.wp4_3_dm262_r_Result_Data_64_bytes_1[44];
	PlcInputs.wp4_3_dm262_r_Result_Data_64_bytes_1[45] := HwInputs.wp4_3_dm262_r_Result_Data_64_bytes_1[45];
	PlcInputs.wp4_3_dm262_r_Result_Data_64_bytes_1[46] := HwInputs.wp4_3_dm262_r_Result_Data_64_bytes_1[46];
	PlcInputs.wp4_3_dm262_r_Result_Data_64_bytes_1[47] := HwInputs.wp4_3_dm262_r_Result_Data_64_bytes_1[47];
	PlcInputs.wp4_3_dm262_r_Result_Data_64_bytes_1[48] := HwInputs.wp4_3_dm262_r_Result_Data_64_bytes_1[48];
	PlcInputs.wp4_3_dm262_r_Result_Data_64_bytes_1[49] := HwInputs.wp4_3_dm262_r_Result_Data_64_bytes_1[49];
	PlcInputs.wp4_3_dm262_r_Result_Data_64_bytes_1[50] := HwInputs.wp4_3_dm262_r_Result_Data_64_bytes_1[50];
	PlcInputs.wp4_3_dm262_r_Result_Data_64_bytes_1[51] := HwInputs.wp4_3_dm262_r_Result_Data_64_bytes_1[51];
	PlcInputs.wp4_3_dm262_r_Result_Data_64_bytes_1[52] := HwInputs.wp4_3_dm262_r_Result_Data_64_bytes_1[52];
	PlcInputs.wp4_3_dm262_r_Result_Data_64_bytes_1[53] := HwInputs.wp4_3_dm262_r_Result_Data_64_bytes_1[53];
	PlcInputs.wp4_3_dm262_r_Result_Data_64_bytes_1[54] := HwInputs.wp4_3_dm262_r_Result_Data_64_bytes_1[54];
	PlcInputs.wp4_3_dm262_r_Result_Data_64_bytes_1[55] := HwInputs.wp4_3_dm262_r_Result_Data_64_bytes_1[55];
	PlcInputs.wp4_3_dm262_r_Result_Data_64_bytes_1[56] := HwInputs.wp4_3_dm262_r_Result_Data_64_bytes_1[56];
	PlcInputs.wp4_3_dm262_r_Result_Data_64_bytes_1[57] := HwInputs.wp4_3_dm262_r_Result_Data_64_bytes_1[57];
	PlcInputs.wp4_3_dm262_r_Result_Data_64_bytes_1[58] := HwInputs.wp4_3_dm262_r_Result_Data_64_bytes_1[58];
	PlcInputs.wp4_3_dm262_r_Result_Data_64_bytes_1[59] := HwInputs.wp4_3_dm262_r_Result_Data_64_bytes_1[59];
	PlcInputs.wp4_3_dm262_r_Result_Data_64_bytes_1[60] := HwInputs.wp4_3_dm262_r_Result_Data_64_bytes_1[60];
	PlcInputs.wp4_3_dm262_r_Result_Data_64_bytes_1[61] := HwInputs.wp4_3_dm262_r_Result_Data_64_bytes_1[61];
	PlcInputs.wp4_3_dm262_r_Result_Data_64_bytes_1[62] := HwInputs.wp4_3_dm262_r_Result_Data_64_bytes_1[62];
	PlcInputs.wp4_3_dm262_r_Result_Data_64_bytes_1[63] := HwInputs.wp4_3_dm262_r_Result_Data_64_bytes_1[63];
	PlcInputs.wp4_3_dm262_r_Result_Data_64_bytes_1[64] := HwInputs.wp4_3_dm262_r_Result_Data_64_bytes_1[64];
	PlcInputs.wp4_3_dm262_r_Result_Data_64_bytes_1[65] := HwInputs.wp4_3_dm262_r_Result_Data_64_bytes_1[65];
	PlcInputs.wp4_3_dm262_r_Result_Data_64_bytes_1[66] := HwInputs.wp4_3_dm262_r_Result_Data_64_bytes_1[66];
	PlcInputs.wp4_3_dm262_r_Result_Data_64_bytes_1[67] := HwInputs.wp4_3_dm262_r_Result_Data_64_bytes_1[67];
	PlcInputs.wp4_3_dm262_r_Result_Data_64_bytes_1[68] := HwInputs.wp4_3_dm262_r_Result_Data_64_bytes_1[68];
	PlcInputs.wp4_3_dm262_r_Result_Data_64_bytes_1[69] := HwInputs.wp4_3_dm262_r_Result_Data_64_bytes_1[69];
	PlcInputs.wp4_3_dm262_r_Result_Data_64_bytes_1[70] := HwInputs.wp4_3_dm262_r_Result_Data_64_bytes_1[70];
	PlcInputs.wp4_3_dm262_r_Result_Data_64_bytes_1[71] := HwInputs.wp4_3_dm262_r_Result_Data_64_bytes_1[71];
END_FUNCTION

(* ---- CopyOutputs.st ---- *)
FUNCTION CopyOutputs
	VAR_EXTERNAL
		HwOutputs : HwOutputs;
		PlcOutputs : PlcOutputs;
	END_VAR
	HwOutputs.wp4_3_dm262_l_Acquisition_Control_1 := PlcOutputs.wp4_3_dm262_l_Acquisition_Control_1;
	HwOutputs.wp4_3_dm262_l_Results_Control_1 := PlcOutputs.wp4_3_dm262_l_Results_Control_1;
	HwOutputs.wp4_3_dm262_l_Soft_Event_Control_1 := PlcOutputs.wp4_3_dm262_l_Soft_Event_Control_1;
	HwOutputs.wp4_3_dm262_l_User_Data_64_bytes_1[0] := PlcOutputs.wp4_3_dm262_l_User_Data_64_bytes_1[0];
	HwOutputs.wp4_3_dm262_l_User_Data_64_bytes_1[1] := PlcOutputs.wp4_3_dm262_l_User_Data_64_bytes_1[1];
	HwOutputs.wp4_3_dm262_l_User_Data_64_bytes_1[2] := PlcOutputs.wp4_3_dm262_l_User_Data_64_bytes_1[2];
	HwOutputs.wp4_3_dm262_l_User_Data_64_bytes_1[3] := PlcOutputs.wp4_3_dm262_l_User_Data_64_bytes_1[3];
	HwOutputs.wp4_3_dm262_l_User_Data_64_bytes_1[4] := PlcOutputs.wp4_3_dm262_l_User_Data_64_bytes_1[4];
	HwOutputs.wp4_3_dm262_l_User_Data_64_bytes_1[5] := PlcOutputs.wp4_3_dm262_l_User_Data_64_bytes_1[5];
	HwOutputs.wp4_3_dm262_l_User_Data_64_bytes_1[6] := PlcOutputs.wp4_3_dm262_l_User_Data_64_bytes_1[6];
	HwOutputs.wp4_3_dm262_l_User_Data_64_bytes_1[7] := PlcOutputs.wp4_3_dm262_l_User_Data_64_bytes_1[7];
	HwOutputs.wp4_3_dm262_l_User_Data_64_bytes_1[8] := PlcOutputs.wp4_3_dm262_l_User_Data_64_bytes_1[8];
	HwOutputs.wp4_3_dm262_l_User_Data_64_bytes_1[9] := PlcOutputs.wp4_3_dm262_l_User_Data_64_bytes_1[9];
	HwOutputs.wp4_3_dm262_l_User_Data_64_bytes_1[10] := PlcOutputs.wp4_3_dm262_l_User_Data_64_bytes_1[10];
	HwOutputs.wp4_3_dm262_l_User_Data_64_bytes_1[11] := PlcOutputs.wp4_3_dm262_l_User_Data_64_bytes_1[11];
	HwOutputs.wp4_3_dm262_l_User_Data_64_bytes_1[12] := PlcOutputs.wp4_3_dm262_l_User_Data_64_bytes_1[12];
	HwOutputs.wp4_3_dm262_l_User_Data_64_bytes_1[13] := PlcOutputs.wp4_3_dm262_l_User_Data_64_bytes_1[13];
	HwOutputs.wp4_3_dm262_l_User_Data_64_bytes_1[14] := PlcOutputs.wp4_3_dm262_l_User_Data_64_bytes_1[14];
	HwOutputs.wp4_3_dm262_l_User_Data_64_bytes_1[15] := PlcOutputs.wp4_3_dm262_l_User_Data_64_bytes_1[15];
	HwOutputs.wp4_3_dm262_l_User_Data_64_bytes_1[16] := PlcOutputs.wp4_3_dm262_l_User_Data_64_bytes_1[16];
	HwOutputs.wp4_3_dm262_l_User_Data_64_bytes_1[17] := PlcOutputs.wp4_3_dm262_l_User_Data_64_bytes_1[17];
	HwOutputs.wp4_3_dm262_l_User_Data_64_bytes_1[18] := PlcOutputs.wp4_3_dm262_l_User_Data_64_bytes_1[18];
	HwOutputs.wp4_3_dm262_l_User_Data_64_bytes_1[19] := PlcOutputs.wp4_3_dm262_l_User_Data_64_bytes_1[19];
	HwOutputs.wp4_3_dm262_l_User_Data_64_bytes_1[20] := PlcOutputs.wp4_3_dm262_l_User_Data_64_bytes_1[20];
	HwOutputs.wp4_3_dm262_l_User_Data_64_bytes_1[21] := PlcOutputs.wp4_3_dm262_l_User_Data_64_bytes_1[21];
	HwOutputs.wp4_3_dm262_l_User_Data_64_bytes_1[22] := PlcOutputs.wp4_3_dm262_l_User_Data_64_bytes_1[22];
	HwOutputs.wp4_3_dm262_l_User_Data_64_bytes_1[23] := PlcOutputs.wp4_3_dm262_l_User_Data_64_bytes_1[23];
	HwOutputs.wp4_3_dm262_l_User_Data_64_bytes_1[24] := PlcOutputs.wp4_3_dm262_l_User_Data_64_bytes_1[24];
	HwOutputs.wp4_3_dm262_l_User_Data_64_bytes_1[25] := PlcOutputs.wp4_3_dm262_l_User_Data_64_bytes_1[25];
	HwOutputs.wp4_3_dm262_l_User_Data_64_bytes_1[26] := PlcOutputs.wp4_3_dm262_l_User_Data_64_bytes_1[26];
	HwOutputs.wp4_3_dm262_l_User_Data_64_bytes_1[27] := PlcOutputs.wp4_3_dm262_l_User_Data_64_bytes_1[27];
	HwOutputs.wp4_3_dm262_l_User_Data_64_bytes_1[28] := PlcOutputs.wp4_3_dm262_l_User_Data_64_bytes_1[28];
	HwOutputs.wp4_3_dm262_l_User_Data_64_bytes_1[29] := PlcOutputs.wp4_3_dm262_l_User_Data_64_bytes_1[29];
	HwOutputs.wp4_3_dm262_l_User_Data_64_bytes_1[30] := PlcOutputs.wp4_3_dm262_l_User_Data_64_bytes_1[30];
	HwOutputs.wp4_3_dm262_l_User_Data_64_bytes_1[31] := PlcOutputs.wp4_3_dm262_l_User_Data_64_bytes_1[31];
	HwOutputs.wp4_3_dm262_l_User_Data_64_bytes_1[32] := PlcOutputs.wp4_3_dm262_l_User_Data_64_bytes_1[32];
	HwOutputs.wp4_3_dm262_l_User_Data_64_bytes_1[33] := PlcOutputs.wp4_3_dm262_l_User_Data_64_bytes_1[33];
	HwOutputs.wp4_3_dm262_l_User_Data_64_bytes_1[34] := PlcOutputs.wp4_3_dm262_l_User_Data_64_bytes_1[34];
	HwOutputs.wp4_3_dm262_l_User_Data_64_bytes_1[35] := PlcOutputs.wp4_3_dm262_l_User_Data_64_bytes_1[35];
	HwOutputs.wp4_3_dm262_l_User_Data_64_bytes_1[36] := PlcOutputs.wp4_3_dm262_l_User_Data_64_bytes_1[36];
	HwOutputs.wp4_3_dm262_l_User_Data_64_bytes_1[37] := PlcOutputs.wp4_3_dm262_l_User_Data_64_bytes_1[37];
	HwOutputs.wp4_3_dm262_l_User_Data_64_bytes_1[38] := PlcOutputs.wp4_3_dm262_l_User_Data_64_bytes_1[38];
	HwOutputs.wp4_3_dm262_l_User_Data_64_bytes_1[39] := PlcOutputs.wp4_3_dm262_l_User_Data_64_bytes_1[39];
	HwOutputs.wp4_3_dm262_l_User_Data_64_bytes_1[40] := PlcOutputs.wp4_3_dm262_l_User_Data_64_bytes_1[40];
	HwOutputs.wp4_3_dm262_l_User_Data_64_bytes_1[41] := PlcOutputs.wp4_3_dm262_l_User_Data_64_bytes_1[41];
	HwOutputs.wp4_3_dm262_l_User_Data_64_bytes_1[42] := PlcOutputs.wp4_3_dm262_l_User_Data_64_bytes_1[42];
	HwOutputs.wp4_3_dm262_l_User_Data_64_bytes_1[43] := PlcOutputs.wp4_3_dm262_l_User_Data_64_bytes_1[43];
	HwOutputs.wp4_3_dm262_l_User_Data_64_bytes_1[44] := PlcOutputs.wp4_3_dm262_l_User_Data_64_bytes_1[44];
	HwOutputs.wp4_3_dm262_l_User_Data_64_bytes_1[45] := PlcOutputs.wp4_3_dm262_l_User_Data_64_bytes_1[45];
	HwOutputs.wp4_3_dm262_l_User_Data_64_bytes_1[46] := PlcOutputs.wp4_3_dm262_l_User_Data_64_bytes_1[46];
	HwOutputs.wp4_3_dm262_l_User_Data_64_bytes_1[47] := PlcOutputs.wp4_3_dm262_l_User_Data_64_bytes_1[47];
	HwOutputs.wp4_3_dm262_l_User_Data_64_bytes_1[48] := PlcOutputs.wp4_3_dm262_l_User_Data_64_bytes_1[48];
	HwOutputs.wp4_3_dm262_l_User_Data_64_bytes_1[49] := PlcOutputs.wp4_3_dm262_l_User_Data_64_bytes_1[49];
	HwOutputs.wp4_3_dm262_l_User_Data_64_bytes_1[50] := PlcOutputs.wp4_3_dm262_l_User_Data_64_bytes_1[50];
	HwOutputs.wp4_3_dm262_l_User_Data_64_bytes_1[51] := PlcOutputs.wp4_3_dm262_l_User_Data_64_bytes_1[51];
	HwOutputs.wp4_3_dm262_l_User_Data_64_bytes_1[52] := PlcOutputs.wp4_3_dm262_l_User_Data_64_bytes_1[52];
	HwOutputs.wp4_3_dm262_l_User_Data_64_bytes_1[53] := PlcOutputs.wp4_3_dm262_l_User_Data_64_bytes_1[53];
	HwOutputs.wp4_3_dm262_l_User_Data_64_bytes_1[54] := PlcOutputs.wp4_3_dm262_l_User_Data_64_bytes_1[54];
	HwOutputs.wp4_3_dm262_l_User_Data_64_bytes_1[55] := PlcOutputs.wp4_3_dm262_l_User_Data_64_bytes_1[55];
	HwOutputs.wp4_3_dm262_l_User_Data_64_bytes_1[56] := PlcOutputs.wp4_3_dm262_l_User_Data_64_bytes_1[56];
	HwOutputs.wp4_3_dm262_l_User_Data_64_bytes_1[57] := PlcOutputs.wp4_3_dm262_l_User_Data_64_bytes_1[57];
	HwOutputs.wp4_3_dm262_l_User_Data_64_bytes_1[58] := PlcOutputs.wp4_3_dm262_l_User_Data_64_bytes_1[58];
	HwOutputs.wp4_3_dm262_l_User_Data_64_bytes_1[59] := PlcOutputs.wp4_3_dm262_l_User_Data_64_bytes_1[59];
	HwOutputs.wp4_3_dm262_l_User_Data_64_bytes_1[60] := PlcOutputs.wp4_3_dm262_l_User_Data_64_bytes_1[60];
	HwOutputs.wp4_3_dm262_l_User_Data_64_bytes_1[61] := PlcOutputs.wp4_3_dm262_l_User_Data_64_bytes_1[61];
	HwOutputs.wp4_3_dm262_l_User_Data_64_bytes_1[62] := PlcOutputs.wp4_3_dm262_l_User_Data_64_bytes_1[62];
	HwOutputs.wp4_3_dm262_l_User_Data_64_bytes_1[63] := PlcOutputs.wp4_3_dm262_l_User_Data_64_bytes_1[63];
	HwOutputs.wp4_3_dm262_l_User_Data_64_bytes_1[64] := PlcOutputs.wp4_3_dm262_l_User_Data_64_bytes_1[64];
	HwOutputs.wp4_3_dm262_l_User_Data_64_bytes_1[65] := PlcOutputs.wp4_3_dm262_l_User_Data_64_bytes_1[65];
	HwOutputs.wp4_3_dm262_l_User_Data_64_bytes_1[66] := PlcOutputs.wp4_3_dm262_l_User_Data_64_bytes_1[66];
	HwOutputs.wp4_3_dm262_l_User_Data_64_bytes_1[67] := PlcOutputs.wp4_3_dm262_l_User_Data_64_bytes_1[67];
	HwOutputs.ET_200SP_ST43_DQ_16x24VDC_0_5A_ST_1 := PlcOutputs.ET_200SP_ST43_DQ_16x24VDC_0_5A_ST_1;
	HwOutputs.ET_200SP_ST43_DQ_16x24VDC_0_5A_ST_2 := PlcOutputs.ET_200SP_ST43_DQ_16x24VDC_0_5A_ST_2;
	HwOutputs.ET_200SP_ST43_TM_Pulse_2x24V_1[0] := PlcOutputs.ET_200SP_ST43_TM_Pulse_2x24V_1[0];
	HwOutputs.ET_200SP_ST43_TM_Pulse_2x24V_1[1] := PlcOutputs.ET_200SP_ST43_TM_Pulse_2x24V_1[1];
	HwOutputs.ET_200SP_ST43_TM_Pulse_2x24V_1[2] := PlcOutputs.ET_200SP_ST43_TM_Pulse_2x24V_1[2];
	HwOutputs.ET_200SP_ST43_TM_Pulse_2x24V_1[3] := PlcOutputs.ET_200SP_ST43_TM_Pulse_2x24V_1[3];
	HwOutputs.ET_200SP_ST43_TM_Pulse_2x24V_1[4] := PlcOutputs.ET_200SP_ST43_TM_Pulse_2x24V_1[4];
	HwOutputs.ET_200SP_ST43_TM_Pulse_2x24V_1[5] := PlcOutputs.ET_200SP_ST43_TM_Pulse_2x24V_1[5];
	HwOutputs.ET_200SP_ST43_TM_Pulse_2x24V_1[6] := PlcOutputs.ET_200SP_ST43_TM_Pulse_2x24V_1[6];
	HwOutputs.ET_200SP_ST43_TM_Pulse_2x24V_1[7] := PlcOutputs.ET_200SP_ST43_TM_Pulse_2x24V_1[7];
	HwOutputs.ET_200SP_ST43_TM_Pulse_2x24V_1[8] := PlcOutputs.ET_200SP_ST43_TM_Pulse_2x24V_1[8];
	HwOutputs.ET_200SP_ST43_TM_Pulse_2x24V_1[9] := PlcOutputs.ET_200SP_ST43_TM_Pulse_2x24V_1[9];
	HwOutputs.ET_200SP_ST43_TM_Pulse_2x24V_1[10] := PlcOutputs.ET_200SP_ST43_TM_Pulse_2x24V_1[10];
	HwOutputs.ET_200SP_ST43_TM_Pulse_2x24V_1[11] := PlcOutputs.ET_200SP_ST43_TM_Pulse_2x24V_1[11];
	HwOutputs.ET_200SP_ST43_TM_Pulse_2x24V_1[12] := PlcOutputs.ET_200SP_ST43_TM_Pulse_2x24V_1[12];
	HwOutputs.ET_200SP_ST43_TM_Pulse_2x24V_1[13] := PlcOutputs.ET_200SP_ST43_TM_Pulse_2x24V_1[13];
	HwOutputs.ET_200SP_ST43_TM_Pulse_2x24V_1[14] := PlcOutputs.ET_200SP_ST43_TM_Pulse_2x24V_1[14];
	HwOutputs.ET_200SP_ST43_TM_Pulse_2x24V_1[15] := PlcOutputs.ET_200SP_ST43_TM_Pulse_2x24V_1[15];
	HwOutputs.ET_200SP_ST43_TM_Pulse_2x24V_1[16] := PlcOutputs.ET_200SP_ST43_TM_Pulse_2x24V_1[16];
	HwOutputs.ET_200SP_ST43_TM_Pulse_2x24V_1[17] := PlcOutputs.ET_200SP_ST43_TM_Pulse_2x24V_1[17];
	HwOutputs.ET_200SP_ST43_TM_Pulse_2x24V_1[18] := PlcOutputs.ET_200SP_ST43_TM_Pulse_2x24V_1[18];
	HwOutputs.ET_200SP_ST43_TM_Pulse_2x24V_1[19] := PlcOutputs.ET_200SP_ST43_TM_Pulse_2x24V_1[19];
	HwOutputs.ET_200SP_ST43_TM_Pulse_2x24V_1[20] := PlcOutputs.ET_200SP_ST43_TM_Pulse_2x24V_1[20];
	HwOutputs.ET_200SP_ST43_TM_Pulse_2x24V_1[21] := PlcOutputs.ET_200SP_ST43_TM_Pulse_2x24V_1[21];
	HwOutputs.ET_200SP_ST43_TM_Pulse_2x24V_1[22] := PlcOutputs.ET_200SP_ST43_TM_Pulse_2x24V_1[22];
	HwOutputs.ET_200SP_ST43_TM_Pulse_2x24V_1[23] := PlcOutputs.ET_200SP_ST43_TM_Pulse_2x24V_1[23];
	HwOutputs.ET_200SP_ST43_TM_Pulse_2x24V_2[0] := PlcOutputs.ET_200SP_ST43_TM_Pulse_2x24V_2[0];
	HwOutputs.ET_200SP_ST43_TM_Pulse_2x24V_2[1] := PlcOutputs.ET_200SP_ST43_TM_Pulse_2x24V_2[1];
	HwOutputs.ET_200SP_ST43_TM_Pulse_2x24V_2[2] := PlcOutputs.ET_200SP_ST43_TM_Pulse_2x24V_2[2];
	HwOutputs.ET_200SP_ST43_TM_Pulse_2x24V_2[3] := PlcOutputs.ET_200SP_ST43_TM_Pulse_2x24V_2[3];
	HwOutputs.ET_200SP_ST43_TM_Pulse_2x24V_2[4] := PlcOutputs.ET_200SP_ST43_TM_Pulse_2x24V_2[4];
	HwOutputs.ET_200SP_ST43_TM_Pulse_2x24V_2[5] := PlcOutputs.ET_200SP_ST43_TM_Pulse_2x24V_2[5];
	HwOutputs.ET_200SP_ST43_TM_Pulse_2x24V_2[6] := PlcOutputs.ET_200SP_ST43_TM_Pulse_2x24V_2[6];
	HwOutputs.ET_200SP_ST43_TM_Pulse_2x24V_2[7] := PlcOutputs.ET_200SP_ST43_TM_Pulse_2x24V_2[7];
	HwOutputs.ET_200SP_ST43_TM_Pulse_2x24V_2[8] := PlcOutputs.ET_200SP_ST43_TM_Pulse_2x24V_2[8];
	HwOutputs.ET_200SP_ST43_TM_Pulse_2x24V_2[9] := PlcOutputs.ET_200SP_ST43_TM_Pulse_2x24V_2[9];
	HwOutputs.ET_200SP_ST43_TM_Pulse_2x24V_2[10] := PlcOutputs.ET_200SP_ST43_TM_Pulse_2x24V_2[10];
	HwOutputs.ET_200SP_ST43_TM_Pulse_2x24V_2[11] := PlcOutputs.ET_200SP_ST43_TM_Pulse_2x24V_2[11];
	HwOutputs.ET_200SP_ST43_TM_Pulse_2x24V_2[12] := PlcOutputs.ET_200SP_ST43_TM_Pulse_2x24V_2[12];
	HwOutputs.ET_200SP_ST43_TM_Pulse_2x24V_2[13] := PlcOutputs.ET_200SP_ST43_TM_Pulse_2x24V_2[13];
	HwOutputs.ET_200SP_ST43_TM_Pulse_2x24V_2[14] := PlcOutputs.ET_200SP_ST43_TM_Pulse_2x24V_2[14];
	HwOutputs.ET_200SP_ST43_TM_Pulse_2x24V_2[15] := PlcOutputs.ET_200SP_ST43_TM_Pulse_2x24V_2[15];
	HwOutputs.ET_200SP_ST43_TM_Pulse_2x24V_2[16] := PlcOutputs.ET_200SP_ST43_TM_Pulse_2x24V_2[16];
	HwOutputs.ET_200SP_ST43_TM_Pulse_2x24V_2[17] := PlcOutputs.ET_200SP_ST43_TM_Pulse_2x24V_2[17];
	HwOutputs.ET_200SP_ST43_TM_Pulse_2x24V_2[18] := PlcOutputs.ET_200SP_ST43_TM_Pulse_2x24V_2[18];
	HwOutputs.ET_200SP_ST43_TM_Pulse_2x24V_2[19] := PlcOutputs.ET_200SP_ST43_TM_Pulse_2x24V_2[19];
	HwOutputs.ET_200SP_ST43_TM_Pulse_2x24V_2[20] := PlcOutputs.ET_200SP_ST43_TM_Pulse_2x24V_2[20];
	HwOutputs.ET_200SP_ST43_TM_Pulse_2x24V_2[21] := PlcOutputs.ET_200SP_ST43_TM_Pulse_2x24V_2[21];
	HwOutputs.ET_200SP_ST43_TM_Pulse_2x24V_2[22] := PlcOutputs.ET_200SP_ST43_TM_Pulse_2x24V_2[22];
	HwOutputs.ET_200SP_ST43_TM_Pulse_2x24V_2[23] := PlcOutputs.ET_200SP_ST43_TM_Pulse_2x24V_2[23];
	HwOutputs.ET_200SP_ST43_TM_Pulse_2x24V_3[0] := PlcOutputs.ET_200SP_ST43_TM_Pulse_2x24V_3[0];
	HwOutputs.ET_200SP_ST43_TM_Pulse_2x24V_3[1] := PlcOutputs.ET_200SP_ST43_TM_Pulse_2x24V_3[1];
	HwOutputs.ET_200SP_ST43_TM_Pulse_2x24V_3[2] := PlcOutputs.ET_200SP_ST43_TM_Pulse_2x24V_3[2];
	HwOutputs.ET_200SP_ST43_TM_Pulse_2x24V_3[3] := PlcOutputs.ET_200SP_ST43_TM_Pulse_2x24V_3[3];
	HwOutputs.ET_200SP_ST43_TM_Pulse_2x24V_3[4] := PlcOutputs.ET_200SP_ST43_TM_Pulse_2x24V_3[4];
	HwOutputs.ET_200SP_ST43_TM_Pulse_2x24V_3[5] := PlcOutputs.ET_200SP_ST43_TM_Pulse_2x24V_3[5];
	HwOutputs.ET_200SP_ST43_TM_Pulse_2x24V_3[6] := PlcOutputs.ET_200SP_ST43_TM_Pulse_2x24V_3[6];
	HwOutputs.ET_200SP_ST43_TM_Pulse_2x24V_3[7] := PlcOutputs.ET_200SP_ST43_TM_Pulse_2x24V_3[7];
	HwOutputs.ET_200SP_ST43_TM_Pulse_2x24V_3[8] := PlcOutputs.ET_200SP_ST43_TM_Pulse_2x24V_3[8];
	HwOutputs.ET_200SP_ST43_TM_Pulse_2x24V_3[9] := PlcOutputs.ET_200SP_ST43_TM_Pulse_2x24V_3[9];
	HwOutputs.ET_200SP_ST43_TM_Pulse_2x24V_3[10] := PlcOutputs.ET_200SP_ST43_TM_Pulse_2x24V_3[10];
	HwOutputs.ET_200SP_ST43_TM_Pulse_2x24V_3[11] := PlcOutputs.ET_200SP_ST43_TM_Pulse_2x24V_3[11];
	HwOutputs.ET_200SP_ST43_TM_Pulse_2x24V_3[12] := PlcOutputs.ET_200SP_ST43_TM_Pulse_2x24V_3[12];
	HwOutputs.ET_200SP_ST43_TM_Pulse_2x24V_3[13] := PlcOutputs.ET_200SP_ST43_TM_Pulse_2x24V_3[13];
	HwOutputs.ET_200SP_ST43_TM_Pulse_2x24V_3[14] := PlcOutputs.ET_200SP_ST43_TM_Pulse_2x24V_3[14];
	HwOutputs.ET_200SP_ST43_TM_Pulse_2x24V_3[15] := PlcOutputs.ET_200SP_ST43_TM_Pulse_2x24V_3[15];
	HwOutputs.ET_200SP_ST43_TM_Pulse_2x24V_3[16] := PlcOutputs.ET_200SP_ST43_TM_Pulse_2x24V_3[16];
	HwOutputs.ET_200SP_ST43_TM_Pulse_2x24V_3[17] := PlcOutputs.ET_200SP_ST43_TM_Pulse_2x24V_3[17];
	HwOutputs.ET_200SP_ST43_TM_Pulse_2x24V_3[18] := PlcOutputs.ET_200SP_ST43_TM_Pulse_2x24V_3[18];
	HwOutputs.ET_200SP_ST43_TM_Pulse_2x24V_3[19] := PlcOutputs.ET_200SP_ST43_TM_Pulse_2x24V_3[19];
	HwOutputs.ET_200SP_ST43_TM_Pulse_2x24V_3[20] := PlcOutputs.ET_200SP_ST43_TM_Pulse_2x24V_3[20];
	HwOutputs.ET_200SP_ST43_TM_Pulse_2x24V_3[21] := PlcOutputs.ET_200SP_ST43_TM_Pulse_2x24V_3[21];
	HwOutputs.ET_200SP_ST43_TM_Pulse_2x24V_3[22] := PlcOutputs.ET_200SP_ST43_TM_Pulse_2x24V_3[22];
	HwOutputs.ET_200SP_ST43_TM_Pulse_2x24V_3[23] := PlcOutputs.ET_200SP_ST43_TM_Pulse_2x24V_3[23];
	HwOutputs.ET_200SP_ST43_TM_Pulse_2x24V_4[0] := PlcOutputs.ET_200SP_ST43_TM_Pulse_2x24V_4[0];
	HwOutputs.ET_200SP_ST43_TM_Pulse_2x24V_4[1] := PlcOutputs.ET_200SP_ST43_TM_Pulse_2x24V_4[1];
	HwOutputs.ET_200SP_ST43_TM_Pulse_2x24V_4[2] := PlcOutputs.ET_200SP_ST43_TM_Pulse_2x24V_4[2];
	HwOutputs.ET_200SP_ST43_TM_Pulse_2x24V_4[3] := PlcOutputs.ET_200SP_ST43_TM_Pulse_2x24V_4[3];
	HwOutputs.ET_200SP_ST43_TM_Pulse_2x24V_4[4] := PlcOutputs.ET_200SP_ST43_TM_Pulse_2x24V_4[4];
	HwOutputs.ET_200SP_ST43_TM_Pulse_2x24V_4[5] := PlcOutputs.ET_200SP_ST43_TM_Pulse_2x24V_4[5];
	HwOutputs.ET_200SP_ST43_TM_Pulse_2x24V_4[6] := PlcOutputs.ET_200SP_ST43_TM_Pulse_2x24V_4[6];
	HwOutputs.ET_200SP_ST43_TM_Pulse_2x24V_4[7] := PlcOutputs.ET_200SP_ST43_TM_Pulse_2x24V_4[7];
	HwOutputs.ET_200SP_ST43_TM_Pulse_2x24V_4[8] := PlcOutputs.ET_200SP_ST43_TM_Pulse_2x24V_4[8];
	HwOutputs.ET_200SP_ST43_TM_Pulse_2x24V_4[9] := PlcOutputs.ET_200SP_ST43_TM_Pulse_2x24V_4[9];
	HwOutputs.ET_200SP_ST43_TM_Pulse_2x24V_4[10] := PlcOutputs.ET_200SP_ST43_TM_Pulse_2x24V_4[10];
	HwOutputs.ET_200SP_ST43_TM_Pulse_2x24V_4[11] := PlcOutputs.ET_200SP_ST43_TM_Pulse_2x24V_4[11];
	HwOutputs.ET_200SP_ST43_TM_Pulse_2x24V_4[12] := PlcOutputs.ET_200SP_ST43_TM_Pulse_2x24V_4[12];
	HwOutputs.ET_200SP_ST43_TM_Pulse_2x24V_4[13] := PlcOutputs.ET_200SP_ST43_TM_Pulse_2x24V_4[13];
	HwOutputs.ET_200SP_ST43_TM_Pulse_2x24V_4[14] := PlcOutputs.ET_200SP_ST43_TM_Pulse_2x24V_4[14];
	HwOutputs.ET_200SP_ST43_TM_Pulse_2x24V_4[15] := PlcOutputs.ET_200SP_ST43_TM_Pulse_2x24V_4[15];
	HwOutputs.ET_200SP_ST43_TM_Pulse_2x24V_4[16] := PlcOutputs.ET_200SP_ST43_TM_Pulse_2x24V_4[16];
	HwOutputs.ET_200SP_ST43_TM_Pulse_2x24V_4[17] := PlcOutputs.ET_200SP_ST43_TM_Pulse_2x24V_4[17];
	HwOutputs.ET_200SP_ST43_TM_Pulse_2x24V_4[18] := PlcOutputs.ET_200SP_ST43_TM_Pulse_2x24V_4[18];
	HwOutputs.ET_200SP_ST43_TM_Pulse_2x24V_4[19] := PlcOutputs.ET_200SP_ST43_TM_Pulse_2x24V_4[19];
	HwOutputs.ET_200SP_ST43_TM_Pulse_2x24V_4[20] := PlcOutputs.ET_200SP_ST43_TM_Pulse_2x24V_4[20];
	HwOutputs.ET_200SP_ST43_TM_Pulse_2x24V_4[21] := PlcOutputs.ET_200SP_ST43_TM_Pulse_2x24V_4[21];
	HwOutputs.ET_200SP_ST43_TM_Pulse_2x24V_4[22] := PlcOutputs.ET_200SP_ST43_TM_Pulse_2x24V_4[22];
	HwOutputs.ET_200SP_ST43_TM_Pulse_2x24V_4[23] := PlcOutputs.ET_200SP_ST43_TM_Pulse_2x24V_4[23];
	HwOutputs.ET_200SP_ST43_TM_Pulse_2x24V_5[0] := PlcOutputs.ET_200SP_ST43_TM_Pulse_2x24V_5[0];
	HwOutputs.ET_200SP_ST43_TM_Pulse_2x24V_5[1] := PlcOutputs.ET_200SP_ST43_TM_Pulse_2x24V_5[1];
	HwOutputs.ET_200SP_ST43_TM_Pulse_2x24V_5[2] := PlcOutputs.ET_200SP_ST43_TM_Pulse_2x24V_5[2];
	HwOutputs.ET_200SP_ST43_TM_Pulse_2x24V_5[3] := PlcOutputs.ET_200SP_ST43_TM_Pulse_2x24V_5[3];
	HwOutputs.ET_200SP_ST43_TM_Pulse_2x24V_5[4] := PlcOutputs.ET_200SP_ST43_TM_Pulse_2x24V_5[4];
	HwOutputs.ET_200SP_ST43_TM_Pulse_2x24V_5[5] := PlcOutputs.ET_200SP_ST43_TM_Pulse_2x24V_5[5];
	HwOutputs.ET_200SP_ST43_TM_Pulse_2x24V_5[6] := PlcOutputs.ET_200SP_ST43_TM_Pulse_2x24V_5[6];
	HwOutputs.ET_200SP_ST43_TM_Pulse_2x24V_5[7] := PlcOutputs.ET_200SP_ST43_TM_Pulse_2x24V_5[7];
	HwOutputs.ET_200SP_ST43_TM_Pulse_2x24V_5[8] := PlcOutputs.ET_200SP_ST43_TM_Pulse_2x24V_5[8];
	HwOutputs.ET_200SP_ST43_TM_Pulse_2x24V_5[9] := PlcOutputs.ET_200SP_ST43_TM_Pulse_2x24V_5[9];
	HwOutputs.ET_200SP_ST43_TM_Pulse_2x24V_5[10] := PlcOutputs.ET_200SP_ST43_TM_Pulse_2x24V_5[10];
	HwOutputs.ET_200SP_ST43_TM_Pulse_2x24V_5[11] := PlcOutputs.ET_200SP_ST43_TM_Pulse_2x24V_5[11];
	HwOutputs.ET_200SP_ST43_TM_Pulse_2x24V_5[12] := PlcOutputs.ET_200SP_ST43_TM_Pulse_2x24V_5[12];
	HwOutputs.ET_200SP_ST43_TM_Pulse_2x24V_5[13] := PlcOutputs.ET_200SP_ST43_TM_Pulse_2x24V_5[13];
	HwOutputs.ET_200SP_ST43_TM_Pulse_2x24V_5[14] := PlcOutputs.ET_200SP_ST43_TM_Pulse_2x24V_5[14];
	HwOutputs.ET_200SP_ST43_TM_Pulse_2x24V_5[15] := PlcOutputs.ET_200SP_ST43_TM_Pulse_2x24V_5[15];
	HwOutputs.ET_200SP_ST43_TM_Pulse_2x24V_5[16] := PlcOutputs.ET_200SP_ST43_TM_Pulse_2x24V_5[16];
	HwOutputs.ET_200SP_ST43_TM_Pulse_2x24V_5[17] := PlcOutputs.ET_200SP_ST43_TM_Pulse_2x24V_5[17];
	HwOutputs.ET_200SP_ST43_TM_Pulse_2x24V_5[18] := PlcOutputs.ET_200SP_ST43_TM_Pulse_2x24V_5[18];
	HwOutputs.ET_200SP_ST43_TM_Pulse_2x24V_5[19] := PlcOutputs.ET_200SP_ST43_TM_Pulse_2x24V_5[19];
	HwOutputs.ET_200SP_ST43_TM_Pulse_2x24V_5[20] := PlcOutputs.ET_200SP_ST43_TM_Pulse_2x24V_5[20];
	HwOutputs.ET_200SP_ST43_TM_Pulse_2x24V_5[21] := PlcOutputs.ET_200SP_ST43_TM_Pulse_2x24V_5[21];
	HwOutputs.ET_200SP_ST43_TM_Pulse_2x24V_5[22] := PlcOutputs.ET_200SP_ST43_TM_Pulse_2x24V_5[22];
	HwOutputs.ET_200SP_ST43_TM_Pulse_2x24V_5[23] := PlcOutputs.ET_200SP_ST43_TM_Pulse_2x24V_5[23];
	HwOutputs.wp4_3_dm262_r_Acquisition_Control_1 := PlcOutputs.wp4_3_dm262_r_Acquisition_Control_1;
	HwOutputs.wp4_3_dm262_r_Results_Control_1 := PlcOutputs.wp4_3_dm262_r_Results_Control_1;
	HwOutputs.wp4_3_dm262_r_Soft_Event_Control_1 := PlcOutputs.wp4_3_dm262_r_Soft_Event_Control_1;
	HwOutputs.wp4_3_dm262_r_User_Data_64_bytes_1[0] := PlcOutputs.wp4_3_dm262_r_User_Data_64_bytes_1[0];
	HwOutputs.wp4_3_dm262_r_User_Data_64_bytes_1[1] := PlcOutputs.wp4_3_dm262_r_User_Data_64_bytes_1[1];
	HwOutputs.wp4_3_dm262_r_User_Data_64_bytes_1[2] := PlcOutputs.wp4_3_dm262_r_User_Data_64_bytes_1[2];
	HwOutputs.wp4_3_dm262_r_User_Data_64_bytes_1[3] := PlcOutputs.wp4_3_dm262_r_User_Data_64_bytes_1[3];
	HwOutputs.wp4_3_dm262_r_User_Data_64_bytes_1[4] := PlcOutputs.wp4_3_dm262_r_User_Data_64_bytes_1[4];
	HwOutputs.wp4_3_dm262_r_User_Data_64_bytes_1[5] := PlcOutputs.wp4_3_dm262_r_User_Data_64_bytes_1[5];
	HwOutputs.wp4_3_dm262_r_User_Data_64_bytes_1[6] := PlcOutputs.wp4_3_dm262_r_User_Data_64_bytes_1[6];
	HwOutputs.wp4_3_dm262_r_User_Data_64_bytes_1[7] := PlcOutputs.wp4_3_dm262_r_User_Data_64_bytes_1[7];
	HwOutputs.wp4_3_dm262_r_User_Data_64_bytes_1[8] := PlcOutputs.wp4_3_dm262_r_User_Data_64_bytes_1[8];
	HwOutputs.wp4_3_dm262_r_User_Data_64_bytes_1[9] := PlcOutputs.wp4_3_dm262_r_User_Data_64_bytes_1[9];
	HwOutputs.wp4_3_dm262_r_User_Data_64_bytes_1[10] := PlcOutputs.wp4_3_dm262_r_User_Data_64_bytes_1[10];
	HwOutputs.wp4_3_dm262_r_User_Data_64_bytes_1[11] := PlcOutputs.wp4_3_dm262_r_User_Data_64_bytes_1[11];
	HwOutputs.wp4_3_dm262_r_User_Data_64_bytes_1[12] := PlcOutputs.wp4_3_dm262_r_User_Data_64_bytes_1[12];
	HwOutputs.wp4_3_dm262_r_User_Data_64_bytes_1[13] := PlcOutputs.wp4_3_dm262_r_User_Data_64_bytes_1[13];
	HwOutputs.wp4_3_dm262_r_User_Data_64_bytes_1[14] := PlcOutputs.wp4_3_dm262_r_User_Data_64_bytes_1[14];
	HwOutputs.wp4_3_dm262_r_User_Data_64_bytes_1[15] := PlcOutputs.wp4_3_dm262_r_User_Data_64_bytes_1[15];
	HwOutputs.wp4_3_dm262_r_User_Data_64_bytes_1[16] := PlcOutputs.wp4_3_dm262_r_User_Data_64_bytes_1[16];
	HwOutputs.wp4_3_dm262_r_User_Data_64_bytes_1[17] := PlcOutputs.wp4_3_dm262_r_User_Data_64_bytes_1[17];
	HwOutputs.wp4_3_dm262_r_User_Data_64_bytes_1[18] := PlcOutputs.wp4_3_dm262_r_User_Data_64_bytes_1[18];
	HwOutputs.wp4_3_dm262_r_User_Data_64_bytes_1[19] := PlcOutputs.wp4_3_dm262_r_User_Data_64_bytes_1[19];
	HwOutputs.wp4_3_dm262_r_User_Data_64_bytes_1[20] := PlcOutputs.wp4_3_dm262_r_User_Data_64_bytes_1[20];
	HwOutputs.wp4_3_dm262_r_User_Data_64_bytes_1[21] := PlcOutputs.wp4_3_dm262_r_User_Data_64_bytes_1[21];
	HwOutputs.wp4_3_dm262_r_User_Data_64_bytes_1[22] := PlcOutputs.wp4_3_dm262_r_User_Data_64_bytes_1[22];
	HwOutputs.wp4_3_dm262_r_User_Data_64_bytes_1[23] := PlcOutputs.wp4_3_dm262_r_User_Data_64_bytes_1[23];
	HwOutputs.wp4_3_dm262_r_User_Data_64_bytes_1[24] := PlcOutputs.wp4_3_dm262_r_User_Data_64_bytes_1[24];
	HwOutputs.wp4_3_dm262_r_User_Data_64_bytes_1[25] := PlcOutputs.wp4_3_dm262_r_User_Data_64_bytes_1[25];
	HwOutputs.wp4_3_dm262_r_User_Data_64_bytes_1[26] := PlcOutputs.wp4_3_dm262_r_User_Data_64_bytes_1[26];
	HwOutputs.wp4_3_dm262_r_User_Data_64_bytes_1[27] := PlcOutputs.wp4_3_dm262_r_User_Data_64_bytes_1[27];
	HwOutputs.wp4_3_dm262_r_User_Data_64_bytes_1[28] := PlcOutputs.wp4_3_dm262_r_User_Data_64_bytes_1[28];
	HwOutputs.wp4_3_dm262_r_User_Data_64_bytes_1[29] := PlcOutputs.wp4_3_dm262_r_User_Data_64_bytes_1[29];
	HwOutputs.wp4_3_dm262_r_User_Data_64_bytes_1[30] := PlcOutputs.wp4_3_dm262_r_User_Data_64_bytes_1[30];
	HwOutputs.wp4_3_dm262_r_User_Data_64_bytes_1[31] := PlcOutputs.wp4_3_dm262_r_User_Data_64_bytes_1[31];
	HwOutputs.wp4_3_dm262_r_User_Data_64_bytes_1[32] := PlcOutputs.wp4_3_dm262_r_User_Data_64_bytes_1[32];
	HwOutputs.wp4_3_dm262_r_User_Data_64_bytes_1[33] := PlcOutputs.wp4_3_dm262_r_User_Data_64_bytes_1[33];
	HwOutputs.wp4_3_dm262_r_User_Data_64_bytes_1[34] := PlcOutputs.wp4_3_dm262_r_User_Data_64_bytes_1[34];
	HwOutputs.wp4_3_dm262_r_User_Data_64_bytes_1[35] := PlcOutputs.wp4_3_dm262_r_User_Data_64_bytes_1[35];
	HwOutputs.wp4_3_dm262_r_User_Data_64_bytes_1[36] := PlcOutputs.wp4_3_dm262_r_User_Data_64_bytes_1[36];
	HwOutputs.wp4_3_dm262_r_User_Data_64_bytes_1[37] := PlcOutputs.wp4_3_dm262_r_User_Data_64_bytes_1[37];
	HwOutputs.wp4_3_dm262_r_User_Data_64_bytes_1[38] := PlcOutputs.wp4_3_dm262_r_User_Data_64_bytes_1[38];
	HwOutputs.wp4_3_dm262_r_User_Data_64_bytes_1[39] := PlcOutputs.wp4_3_dm262_r_User_Data_64_bytes_1[39];
	HwOutputs.wp4_3_dm262_r_User_Data_64_bytes_1[40] := PlcOutputs.wp4_3_dm262_r_User_Data_64_bytes_1[40];
	HwOutputs.wp4_3_dm262_r_User_Data_64_bytes_1[41] := PlcOutputs.wp4_3_dm262_r_User_Data_64_bytes_1[41];
	HwOutputs.wp4_3_dm262_r_User_Data_64_bytes_1[42] := PlcOutputs.wp4_3_dm262_r_User_Data_64_bytes_1[42];
	HwOutputs.wp4_3_dm262_r_User_Data_64_bytes_1[43] := PlcOutputs.wp4_3_dm262_r_User_Data_64_bytes_1[43];
	HwOutputs.wp4_3_dm262_r_User_Data_64_bytes_1[44] := PlcOutputs.wp4_3_dm262_r_User_Data_64_bytes_1[44];
	HwOutputs.wp4_3_dm262_r_User_Data_64_bytes_1[45] := PlcOutputs.wp4_3_dm262_r_User_Data_64_bytes_1[45];
	HwOutputs.wp4_3_dm262_r_User_Data_64_bytes_1[46] := PlcOutputs.wp4_3_dm262_r_User_Data_64_bytes_1[46];
	HwOutputs.wp4_3_dm262_r_User_Data_64_bytes_1[47] := PlcOutputs.wp4_3_dm262_r_User_Data_64_bytes_1[47];
	HwOutputs.wp4_3_dm262_r_User_Data_64_bytes_1[48] := PlcOutputs.wp4_3_dm262_r_User_Data_64_bytes_1[48];
	HwOutputs.wp4_3_dm262_r_User_Data_64_bytes_1[49] := PlcOutputs.wp4_3_dm262_r_User_Data_64_bytes_1[49];
	HwOutputs.wp4_3_dm262_r_User_Data_64_bytes_1[50] := PlcOutputs.wp4_3_dm262_r_User_Data_64_bytes_1[50];
	HwOutputs.wp4_3_dm262_r_User_Data_64_bytes_1[51] := PlcOutputs.wp4_3_dm262_r_User_Data_64_bytes_1[51];
	HwOutputs.wp4_3_dm262_r_User_Data_64_bytes_1[52] := PlcOutputs.wp4_3_dm262_r_User_Data_64_bytes_1[52];
	HwOutputs.wp4_3_dm262_r_User_Data_64_bytes_1[53] := PlcOutputs.wp4_3_dm262_r_User_Data_64_bytes_1[53];
	HwOutputs.wp4_3_dm262_r_User_Data_64_bytes_1[54] := PlcOutputs.wp4_3_dm262_r_User_Data_64_bytes_1[54];
	HwOutputs.wp4_3_dm262_r_User_Data_64_bytes_1[55] := PlcOutputs.wp4_3_dm262_r_User_Data_64_bytes_1[55];
	HwOutputs.wp4_3_dm262_r_User_Data_64_bytes_1[56] := PlcOutputs.wp4_3_dm262_r_User_Data_64_bytes_1[56];
	HwOutputs.wp4_3_dm262_r_User_Data_64_bytes_1[57] := PlcOutputs.wp4_3_dm262_r_User_Data_64_bytes_1[57];
	HwOutputs.wp4_3_dm262_r_User_Data_64_bytes_1[58] := PlcOutputs.wp4_3_dm262_r_User_Data_64_bytes_1[58];
	HwOutputs.wp4_3_dm262_r_User_Data_64_bytes_1[59] := PlcOutputs.wp4_3_dm262_r_User_Data_64_bytes_1[59];
	HwOutputs.wp4_3_dm262_r_User_Data_64_bytes_1[60] := PlcOutputs.wp4_3_dm262_r_User_Data_64_bytes_1[60];
	HwOutputs.wp4_3_dm262_r_User_Data_64_bytes_1[61] := PlcOutputs.wp4_3_dm262_r_User_Data_64_bytes_1[61];
	HwOutputs.wp4_3_dm262_r_User_Data_64_bytes_1[62] := PlcOutputs.wp4_3_dm262_r_User_Data_64_bytes_1[62];
	HwOutputs.wp4_3_dm262_r_User_Data_64_bytes_1[63] := PlcOutputs.wp4_3_dm262_r_User_Data_64_bytes_1[63];
	HwOutputs.wp4_3_dm262_r_User_Data_64_bytes_1[64] := PlcOutputs.wp4_3_dm262_r_User_Data_64_bytes_1[64];
	HwOutputs.wp4_3_dm262_r_User_Data_64_bytes_1[65] := PlcOutputs.wp4_3_dm262_r_User_Data_64_bytes_1[65];
	HwOutputs.wp4_3_dm262_r_User_Data_64_bytes_1[66] := PlcOutputs.wp4_3_dm262_r_User_Data_64_bytes_1[66];
	HwOutputs.wp4_3_dm262_r_User_Data_64_bytes_1[67] := PlcOutputs.wp4_3_dm262_r_User_Data_64_bytes_1[67];
	HwOutputs.CPX_ST43_MPA1S_VMPA1_FB_EMS_8_8DO_1 := PlcOutputs.CPX_ST43_MPA1S_VMPA1_FB_EMS_8_8DO_1;
	HwOutputs.CPX_ST43_MPA1G_VMPA1_FB_EMG_8_8DO_1 := PlcOutputs.CPX_ST43_MPA1G_VMPA1_FB_EMG_8_8DO_1;
	HwOutputs.CPX_ST43_MPA1G_VMPA1_FB_EMG_8_8DO_2 := PlcOutputs.CPX_ST43_MPA1G_VMPA1_FB_EMG_8_8DO_2;
	HwOutputs.CPX_ST43_MPA1G_VMPA1_FB_EMG_8_8DO_3 := PlcOutputs.CPX_ST43_MPA1G_VMPA1_FB_EMG_8_8DO_3;
	HwOutputs.CPX_ST43_MPA1G_VMPA1_FB_EMG_8_8DO_4 := PlcOutputs.CPX_ST43_MPA1G_VMPA1_FB_EMG_8_8DO_4;
	HwOutputs.CPX_ST43_MPA1G_VMPA1_FB_EMG_8_8DO_5 := PlcOutputs.CPX_ST43_MPA1G_VMPA1_FB_EMG_8_8DO_5;
END_FUNCTION
